(* CODESYS project SkyP_crashtest

Project tree, tasks and I/O mapping:
  Device : CODESYS Control for Linux SL, CODESYS, order no. 2302000005, version 4.13.0.0
    Ethernet : Ethernet, CODESYS, version 4.2.0.0
        settings: IPAddress = [192,168,1,12]; SubnetMask = [255,255,255,0]; GatewayAddress = [192,168,1,1]; MACAddress = [16#00,16#E0,16#4F,16#68,16#EC,16#5C]; NetworkInterfaceName = 'eno1'; NetworkInterfaceName = "eno1"; SaveCommunicationSettings = FALSE; IPAddress = [192,168,0,2]; SubnetMask = [255,255,255,0]; GatewayAddress = [0,0,0,0]
      Modbus_TCP_Master : Modbus TCP Client, CODESYS, version 4.4.0.0
          settings: AutoReconnect = TRUE
        Modbus_TCP_Slave_AC1 : Modbus TCP Slave, 3S - Smart Software Solutions GmbH, version 4.1.0.0
            settings: Unit-ID = 255; IPAddress = [192, 168, 0, 51]; Channel 0.Function Code = 3; Channel 0.Read Offset = 16#0000; Channel 0.Read Length = 124; Channel 0.Write Offset = 0; Channel 0.Write Length = 0; Channel 0.Cycle Time = 100; Channel 1.Function Code = 3; Channel 1.Read Offset = 16#007C; Channel 1.Read Length = 124; Channel 1.Write Offset = 0; Channel 1.Write Length = 0; Channel 1.Cycle Time = 100; Channel 2.Function Code = 3; Channel 2.Read Offset = 16#00F8; Channel 2.Read Length = 124; Channel 2.Write Offset = 0; Channel 2.Write Length = 0; Channel 2.Cycle Time = 100; Channel 3.Function Code = 16; Channel 3.Read Offset = 0; Channel 3.Read Length = 0; Channel 3.Write Offset = 16#0114; Channel 3.Write Length = 4; Channel 3.Cycle Time = 100
            input  Application.Chiller_1.modbus_var_1000 : ARRAY[0..123] OF WORD  // Channel 0
            input  Application.Chiller_1.modbus_var_1001 : ARRAY[0..123] OF WORD  // Channel 1
            input  Application.Chiller_1.modbus_var_1002 : ARRAY[0..123] OF WORD  // Channel 2
            output Application.Chiller_1.modbus_var_1002[276] : WORD  // Channel 3.Channel 3
            output Application.Chiller_1.modbus_var_1002[277] : WORD  // Channel 3.Channel 3
            output Application.Chiller_1.modbus_var_1002[278] : WORD  // Channel 3.Channel 3
            output Application.Chiller_1.modbus_var_1002[279] : WORD  // Channel 3.Channel 3
            unmapped channels: Channel 3
        Modbus_TCP_Slave_AC2 : Modbus TCP Slave, 3S - Smart Software Solutions GmbH, version 4.1.0.0
            settings: Unit-ID = 255; IPAddress = [192, 168, 0, 52]; Channel 0.Function Code = 3; Channel 0.Read Offset = 16#0000; Channel 0.Read Length = 124; Channel 0.Write Offset = 0; Channel 0.Write Length = 0; Channel 0.Cycle Time = 100; Channel 1.Function Code = 3; Channel 1.Read Offset = 16#007C; Channel 1.Read Length = 124; Channel 1.Write Offset = 0; Channel 1.Write Length = 0; Channel 1.Cycle Time = 100; Channel 2.Function Code = 3; Channel 2.Read Offset = 16#00F8; Channel 2.Read Length = 124; Channel 2.Write Offset = 0; Channel 2.Write Length = 0; Channel 2.Cycle Time = 100; Channel 3.Function Code = 16; Channel 3.Read Offset = 0; Channel 3.Read Length = 0; Channel 3.Write Offset = 16#0114; Channel 3.Write Length = 4; Channel 3.Cycle Time = 100
            input  Application.Chiller_2.modbus_var_1000 : ARRAY[0..123] OF WORD  // Channel 0
            input  Application.Chiller_2.modbus_var_1001 : ARRAY[0..123] OF WORD  // Channel 1
            input  Application.Chiller_2.modbus_var_1002 : ARRAY[0..123] OF WORD  // Channel 2
            output Application.Chiller_2.modbus_var_1002[276] : WORD  // Channel 3.Channel 3
            output Application.Chiller_2.modbus_var_1002[277] : WORD  // Channel 3.Channel 3
            output Application.Chiller_2.modbus_var_1002[278] : WORD  // Channel 3.Channel 3
            output Application.Chiller_2.modbus_var_1002[279] : WORD  // Channel 3.Channel 3
            unmapped channels: Channel 3
        Modbus_TCP_Slave_AC3 : Modbus TCP Slave, 3S - Smart Software Solutions GmbH, version 4.1.0.0
            settings: Unit-ID = 255; IPAddress = [192, 168, 0, 53]; Channel 0.Function Code = 3; Channel 0.Read Offset = 16#0000; Channel 0.Read Length = 124; Channel 0.Write Offset = 0; Channel 0.Write Length = 0; Channel 0.Cycle Time = 100; Channel 1.Function Code = 3; Channel 1.Read Offset = 16#007C; Channel 1.Read Length = 124; Channel 1.Write Offset = 0; Channel 1.Write Length = 0; Channel 1.Cycle Time = 100; Channel 2.Function Code = 3; Channel 2.Read Offset = 16#00F8; Channel 2.Read Length = 124; Channel 2.Write Offset = 0; Channel 2.Write Length = 0; Channel 2.Cycle Time = 100; Channel 3.Function Code = 16; Channel 3.Read Offset = 0; Channel 3.Read Length = 0; Channel 3.Write Offset = 16#0114; Channel 3.Write Length = 4; Channel 3.Cycle Time = 100
            input  Application.Chiller_3.modbus_var_1000 : ARRAY[0..123] OF WORD  // Channel 0
            input  Application.Chiller_3.modbus_var_1001 : ARRAY[0..123] OF WORD  // Channel 1
            input  Application.Chiller_3.modbus_var_1002 : ARRAY[0..123] OF WORD  // Channel 2
            output Application.Chiller_3.modbus_var_1002[276] : WORD  // Channel 3.Channel 3
            output Application.Chiller_3.modbus_var_1002[277] : WORD  // Channel 3.Channel 3
            output Application.Chiller_3.modbus_var_1002[278] : WORD  // Channel 3.Channel 3
            output Application.Chiller_3.modbus_var_1002[279] : WORD  // Channel 3.Channel 3
            unmapped channels: Channel 3
        Modbus_TCP_Slave_AC4 : Modbus TCP Slave, 3S - Smart Software Solutions GmbH, version 4.1.0.0
            settings: Unit-ID = 255; IPAddress = [192, 168, 0, 54]; Channel 0.Function Code = 3; Channel 0.Read Offset = 16#0000; Channel 0.Read Length = 124; Channel 0.Write Offset = 0; Channel 0.Write Length = 0; Channel 0.Cycle Time = 100; Channel 1.Function Code = 3; Channel 1.Read Offset = 16#007C; Channel 1.Read Length = 124; Channel 1.Write Offset = 0; Channel 1.Write Length = 0; Channel 1.Cycle Time = 100; Channel 2.Function Code = 3; Channel 2.Read Offset = 16#00F8; Channel 2.Read Length = 124; Channel 2.Write Offset = 0; Channel 2.Write Length = 0; Channel 2.Cycle Time = 100; Channel 3.Function Code = 16; Channel 3.Read Offset = 0; Channel 3.Read Length = 0; Channel 3.Write Offset = 16#0114; Channel 3.Write Length = 4; Channel 3.Cycle Time = 100
            input  Application.Chiller_4.modbus_var_1000 : ARRAY[0..123] OF WORD  // Channel 0
            input  Application.Chiller_4.modbus_var_1001 : ARRAY[0..123] OF WORD  // Channel 1
            input  Application.Chiller_4.modbus_var_1002 : ARRAY[0..123] OF WORD  // Channel 2
            output Application.Chiller_4.modbus_var_1002[276] : WORD  // Channel 3.Channel 3
            output Application.Chiller_4.modbus_var_1002[277] : WORD  // Channel 3.Channel 3
            output Application.Chiller_4.modbus_var_1002[278] : WORD  // Channel 3.Channel 3
            output Application.Chiller_4.modbus_var_1002[279] : WORD  // Channel 3.Channel 3
            unmapped channels: Channel 3
        Modbus_TCP_Slave_AC5 : Modbus TCP Slave, 3S - Smart Software Solutions GmbH, version 4.1.0.0
            settings: Unit-ID = 255; IPAddress = [192, 168, 0, 55]; Channel 0.Function Code = 3; Channel 0.Read Offset = 16#0000; Channel 0.Read Length = 124; Channel 0.Write Offset = 0; Channel 0.Write Length = 0; Channel 0.Cycle Time = 100; Channel 1.Function Code = 3; Channel 1.Read Offset = 16#007C; Channel 1.Read Length = 124; Channel 1.Write Offset = 0; Channel 1.Write Length = 0; Channel 1.Cycle Time = 100; Channel 2.Function Code = 3; Channel 2.Read Offset = 16#00F8; Channel 2.Read Length = 124; Channel 2.Write Offset = 0; Channel 2.Write Length = 0; Channel 2.Cycle Time = 100; Channel 3.Function Code = 16; Channel 3.Read Offset = 0; Channel 3.Read Length = 0; Channel 3.Write Offset = 16#0114; Channel 3.Write Length = 4; Channel 3.Cycle Time = 100
            input  Application.Chiller_5.modbus_var_1000 : ARRAY[0..123] OF WORD  // Channel 0
            input  Application.Chiller_5.modbus_var_1001 : ARRAY[0..123] OF WORD  // Channel 1
            input  Application.Chiller_5.modbus_var_1002 : ARRAY[0..123] OF WORD  // Channel 2
            output Application.Chiller_5.modbus_var_1002[276] : WORD  // Channel 3.Channel 3
            output Application.Chiller_5.modbus_var_1002[277] : WORD  // Channel 3.Channel 3
            output Application.Chiller_5.modbus_var_1002[278] : WORD  // Channel 3.Channel 3
            output Application.Chiller_5.modbus_var_1002[279] : WORD  // Channel 3.Channel 3
            unmapped channels: Channel 3
  libraries: CmpBitmapPool, 3.5.17.0 (System); AC_DataLog, 3.5.16.0 (3S - Smart Software Solutions GmbH)
  5ce3da45-db07-42e7-a21c-a00fff4ed8f6|C:\Users\Technician\Desktop\Images\Chiller\Compressor2.png
  5ce3da45-db07-42e7-a21c-a00fff4ed8f6|C:\Users\Technician\Desktop\Images\Chiller\Ejector.png
  5ce3da45-db07-42e7-a21c-a00fff4ed8f6|C:\Users\Technician\Desktop\Images\Chiller\Evaporator2.png
  5ce3da45-db07-42e7-a21c-a00fff4ed8f6|C:\Users\Technician\Desktop\Images\Chiller\OilFilter.png
  5ce3da45-db07-42e7-a21c-a00fff4ed8f6|C:\Users\Technician\Desktop\Images\Chiller\OilReceiver.png
  5ce3da45-db07-42e7-a21c-a00fff4ed8f6|C:\Users\Technician\Desktop\Images\Div bilder\Arrow black down.png
  5ce3da45-db07-42e7-a21c-a00fff4ed8f6|C:\Users\Technician\Desktop\Images\Div bilder\Arrow black left.png
  5ce3da45-db07-42e7-a21c-a00fff4ed8f6|C:\Users\Technician\Desktop\Images\Div bilder\Arrow black right.png
  5ce3da45-db07-42e7-a21c-a00fff4ed8f6|C:\Users\Technician\Desktop\Images\Div bilder\Arrow black up.png
  5ce3da45-db07-42e7-a21c-a00fff4ed8f6|C:\Users\Technician\Desktop\Images\Div bilder\Arrow gray right.png
  5ce3da45-db07-42e7-a21c-a00fff4ed8f6|C:\Users\Technician\Desktop\Images\Div bilder\Arrow red up.png
  5ce3da45-db07-42e7-a21c-a00fff4ed8f6|C:\Users\Technician\Desktop\Images\HeatExchanger\OilHeatExchanger.png
  5ce3da45-db07-42e7-a21c-a00fff4ed8f6|C:\Users\Technician\Desktop\Images\Menu\CalendarIcon.png
  5ce3da45-db07-42e7-a21c-a00fff4ed8f6|C:\Users\Technician\Desktop\Images\Menu\Logo-Carnival.png
  5ce3da45-db07-42e7-a21c-a00fff4ed8f6|C:\Users\Technician\Desktop\Images\Menu\MenuTrends.png
  5ce3da45-db07-42e7-a21c-a00fff4ed8f6|C:\Users\Technician\Desktop\Images\New\VSD_rev2.png
  5ce3da45-db07-42e7-a21c-a00fff4ed8f6|C:\Users\Technician\Desktop\Images\Pipes\PipeBlack_1_Horizontal.png
  5ce3da45-db07-42e7-a21c-a00fff4ed8f6|C:\Users\Technician\Desktop\Images\Pipes\PipeBlack_1_LD.png
  5ce3da45-db07-42e7-a21c-a00fff4ed8f6|C:\Users\Technician\Desktop\Images\Pipes\PipeBlack_1_LU.png
  5ce3da45-db07-42e7-a21c-a00fff4ed8f6|C:\Users\Technician\Desktop\Images\Pipes\PipeBlack_1_RD.png
  5ce3da45-db07-42e7-a21c-a00fff4ed8f6|C:\Users\Technician\Desktop\Images\Pipes\PipeBlack_1_RU.png
  5ce3da45-db07-42e7-a21c-a00fff4ed8f6|C:\Users\Technician\Desktop\Images\Pipes\PipeBlack_1_Vertical.png
  5ce3da45-db07-42e7-a21c-a00fff4ed8f6|C:\Users\Technician\Desktop\Images\Pipes\PipeBlack_1S_H_Faded.png
  5ce3da45-db07-42e7-a21c-a00fff4ed8f6|C:\Users\Technician\Desktop\Images\Ships\Norwegian Prima.jpg
  5ce3da45-db07-42e7-a21c-a00fff4ed8f6|C:\Users\Technician\Desktop\Images\Ships\SkyPrincess.jpg
  5ce3da45-db07-42e7-a21c-a00fff4ed8f6|C:\Users\Technician\Desktop\Images\Valves\RegValve.png
  AC_GENERATOR_DATA
  DataLogManager
    Channels for DataLog (DataLogChannels)
      DataLogChannel_1
        A storage module. (DataLogStorage)
        DataLogStorage_CSV
      DataLogChannel_2
        A storage module. (DataLogStorage)
        DataLogStorage_CSV
      DataLogChannel_3
        A storage module. (DataLogStorage)
        DataLogStorage_CSV
      DataLogChannel_4
        A storage module. (DataLogStorage)
        DataLogStorage_CSV
      DataLogChannel_5
        A storage module. (DataLogStorage)
        DataLogStorage_CSV
      DataLogChannel
        A storage module. (DataLogStorage)
        DataLogStorage_CSV
  text list GlobalTextList
  PersistenceManager
    Channels (pChannels)
      PersistenceChannel
  Alarm Configuration
  visualisation Alarm_list
  program BlinkingAlarm [CFC]
  program Calculus [ST]
  visualisation Chiller1Menu
  visualisation Chiller2Menu
  visualisation Chiller3Menu
  visualisation Chiller4Menu
  visualisation Chiller5Menu
  program Chiller_1 [ST]
  visualisation Chiller_1_Alarm
  visualisation Chiller_1_Flow_Diagram
  visualisation Chiller_1_Oil
  visualisation Chiller_1_Trip
  visualisation Chiller_1_Values
  visualisation Chiller_2_Alarm
  program Chiller_2 [ST]
  visualisation Chiller_2_Flow_Diagram
  visualisation Chiller_2_Oil
  visualisation Chiller_2_Trip
  visualisation Chiller_2_Values
  visualisation Chiller_2_VFD
  program Chiller_3 [ST]
  visualisation Chiller_3_Alarm
  visualisation Chiller_3_Flow_Diagram
  visualisation Chiller_3_Oil
  program Chiller_4 [ST]
  program Chiller_5 [ST]
  text list Chiller_trendvalues
  text list Chiller_VSD_trendvalues
  program csvRead [CFC]
  global variables GVL
  visualisation Homepage
  text list TextList_Local_IAMCS
*)

// GVL
{attribute 'qualified_only'}
VAR_GLOBAL
	COPcalc_data	: ARRAY[0..2, 0..320] OF STRING(100);
	calc_data		: ARRAY[0..8, 0..80] OF STRING(100) ;
	{attribute 'ac_persist' := 'PersistenceChannel'}
	saCOPDataArray			: ARRAY[0..2, 0..320] OF STRING(100);
	{attribute 'ac_persist' := 'PersistenceChannel'}
	saDataArray			: ARRAY[0..8, 0..80] OF STRING(100);
	{attribute 'ac_persist' := 'PersistenceChannel'}
	saDataArray1			: ARRAY[0..8, 0..80] OF STRING(100);
	{attribute 'ac_persist' := 'PersistenceChannel'}
	saDataArray2		: ARRAY[0..8, 0..80] OF STRING(100);
	{attribute 'ac_persist' := 'PersistenceChannel'}
	saDataArray3		: ARRAY[0..8, 0..80] OF STRING(100);
	initRead : BOOL;
	xRead : BOOL;
	xRead1 : BOOL;
	xRead2 : BOOL;
	xRead3 : BOOL;
	xReadCOP : BOOL := FALSE;
	startUp : BOOL;
	presstimer  : TON;
	presstimer2 : TON;
	presstimer3 : TON;
	presstimer4 : TON;
	presstimer5 : TON;
	delaytimer  : TON;
	starttimer1 : BOOL := FALSE  ;
	starttimer2 : BOOL := FALSE  ;
	starttimer3 : BOOL := FALSE  ;
	starttimer4 : BOOL := FALSE  ;
	starttimer5 : BOOL := FALSE  ;
	startdelaytimer : BOOL := FALSE ;
	Startonce : BOOL := FALSE ;
	Startsecond : BOOL := FALSE ;
	{attribute 'ac_persist' := 'PersistenceChannel'}
	PIexpireDate : DATE_AND_TIME := DT#2026-01-31-00:00:00;
	CurrentDate : DATE_AND_TIME ;

END_VAR

// BlinkingAlarm
PROGRAM BlinkingAlarm
VAR
	TimeOn: TIME:= T#1S;
	TimeOff: TIME:= T#1S;
	Alarm: BOOL;
	TurnOn: BOOL;
		
	Blink_0: BLINK;
	
END_VAR
VAR // added by the converter: edge detectors and wires of the graphical bodies
    _w1, _w2 : BOOL;
END_VAR

TurnOn := _w1;
_w1 := not.Sequence.Alarm_sequence OR not.Chiller_1.Unit_alarm OR not.Chiller_1.Unit_trip OR not.Chiller_2.Unit_alarm OR not.Chiller_2.Unit_trip OR not.Chiller_3.Unit_alarm OR not.Chiller_3.Unit_trip OR not.Chiller_4.Unit_alarm OR not.Chiller_4.Unit_trip OR not.Chiller_5.Unit_alarm OR not.Chiller_5.Unit_trip;
_w2 := TurnOn AND Blink_0.OUT;
Blink_0(ENABLE := TurnOn, TIMELOW := TimeOff, TIMEHIGH := TimeOn); // BLINK
Alarm := _w2;

END_PROGRAM

// Chiller_5
PROGRAM Chiller_5
VAR

timer2 : standard.ton ;
{attribute 'ac_datalog_set_default_group' := 'DataLogChannel_5'}
instStruct : LogStruct;


modbus_var : ARRAY[0..100] OF INT;
modbus_var_1000 : ARRAY[0..123] OF WORD;
modbus_var_1001 : ARRAY[124..247] OF WORD;
modbus_var_1002 : ARRAY[248..371] OF WORD;
{attribute 'ac_datalog_hysteresis' := '0.2'}
{attribute 'ac_datalog' := 'DataLogChannel_5'}
Temp_chilled_medium_out : REAL;
{attribute 'ac_datalog_hysteresis' := '0.2'}
{attribute 'ac_datalog' := 'DataLogChannel_5'}
Temp_chilled_medium_in : REAL;
{attribute 'ac_datalog_hysteresis' := '0.2'}
{attribute 'ac_datalog' := 'DataLogChannel_5'}
Temp_water_inlet_cond : REAL;
{attribute 'ac_datalog_hysteresis' := '0.2'}
{attribute 'ac_datalog' := 'DataLogChannel_5'}
Press_suction_compr : REAL;
{attribute 'ac_datalog_hysteresis' := '0.5'}
{attribute 'ac_datalog' := 'DataLogChannel_5'}
Press_discharge_compr : REAL;
{attribute 'ac_datalog_hysteresis' := '0.5'}
{attribute 'ac_datalog' := 'DataLogChannel_5'}
Press_oil_receiver : REAL;
{attribute 'ac_datalog_hysteresis' := '0.5'}
{attribute 'ac_datalog' := 'DataLogChannel_5'}
Press_oil_compr : REAL;
{attribute 'ac_datalog_hysteresis' := '0.4'}
{attribute 'ac_datalog' := 'DataLogChannel_5'}
Temp_discharge : REAL;
{attribute 'ac_datalog_hysteresis' := '0.5'}
{attribute 'ac_datalog' := 'DataLogChannel_5'}
Oil_temp_receiver : REAL;
{attribute 'ac_datalog_hysteresis' := '0.5'}
{attribute 'ac_datalog' := 'DataLogChannel_5'}
Max_motor_temp : REAL;
{attribute 'ac_datalog_hysteresis' := '0.2'}
{attribute 'ac_datalog' := 'DataLogChannel_5'}
Temp_motor_bearing_DE : REAL;
{attribute 'ac_datalog_hysteresis' := '0.2'}
{attribute 'ac_datalog' := 'DataLogChannel_5'}
Temp_motor_bearing_NDE : REAL;
{attribute 'ac_datalog_hysteresis' := '4'}
{attribute 'ac_datalog' := 'DataLogChannel_5'}
Motor_current : REAL;
{attribute 'ac_datalog_hysteresis' := '50'}
{attribute 'ac_datalog' := 'DataLogChannel_5'}
Running_hours_comp_unscaled : WORD;
{attribute 'ac_datalog_hysteresis' := '50'}
{attribute 'ac_datalog' := 'DataLogChannel_5'}
Running_hours_oil_pump_unscaled : WORD;
{attribute 'ac_datalog' := 'DataLogChannel_5'}
Anti_recycle_time : REAL;
{attribute 'ac_datalog_hysteresis' := '2'}
{attribute 'ac_datalog' := 'DataLogChannel_5'}
Feedback_compressor : REAL;
{attribute 'ac_datalog_hysteresis' := '0.2'}
{attribute 'ac_datalog' := 'DataLogChannel_5'}
Oil_diff_pressure : REAL;
{attribute 'ac_datalog_hysteresis' := '0.3'}
{attribute 'ac_datalog' := 'DataLogChannel_5'}
Suction_saturated_temp : REAL;
{attribute 'ac_datalog_hysteresis' := '0.2'}
{attribute 'ac_datalog' := 'DataLogChannel_5'}
Discharge_saturated_temp : REAL;
{attribute 'ac_datalog_hysteresis' := '0.2'}
{attribute 'ac_datalog' := 'DataLogChannel_5'}
Temp_water_outlet_cond : REAL;
{attribute 'ac_datalog_hysteresis' := '0.2'}
{attribute 'ac_datalog' := 'DataLogChannel_5'}
Temp_motor_wind_R : REAL;
{attribute 'ac_datalog_hysteresis' := '0.2'}
{attribute 'ac_datalog' := 'DataLogChannel_5'}
Temp_motor_wind_S : REAL;
{attribute 'ac_datalog_hysteresis' := '0.2'}
{attribute 'ac_datalog' := 'DataLogChannel_5'}
Temp_motor_wind_T : REAL;
{attribute 'ac_datalog_hysteresis' := '0.2'}
{attribute 'ac_datalog' := 'DataLogChannel_5'}
Temp_motor_air : REAL;
{attribute 'ac_datalog_hysteresis' := '0.04'}
{attribute 'ac_datalog' := 'DataLogChannel_5'}
dP_CW : REAL;
{attribute 'ac_datalog_hysteresis' := '0.04'}
{attribute 'ac_datalog' := 'DataLogChannel_5'}
dP_SW : REAL;
{attribute 'ac_datalog_hysteresis' := '4'}
{attribute 'ac_datalog' := 'DataLogChannel_5'}
Chiller_capacity : REAL;
{attribute 'ac_datalog_hysteresis' := '2'}
{attribute 'ac_datalog' := 'DataLogChannel_5'}
Temp_oil_inlet_compr : REAL;
Spare : REAL;
{attribute 'ac_datalog_hysteresis' := '2'}
{attribute 'ac_datalog' := 'DataLogChannel_5'}
SP_CW_controller : REAL;
{attribute 'ac_datalog_hysteresis' := '2'}
{attribute 'ac_datalog' := 'DataLogChannel_5'}
Setpoint_oil_pump : REAL;
{attribute 'ac_datalog_hysteresis' := '0.02'}
{attribute 'ac_datalog' := 'DataLogChannel_5'}
Thrust_bearing_position : REAL;
{attribute 'ac_datalog_hysteresis' := '50'}
{attribute 'ac_datalog' := 'DataLogChannel_5'}
Oil_pump_running_hours : REAL;
{attribute 'ac_datalog_hysteresis' := '5'}
{attribute 'ac_datalog' := 'DataLogChannel_5'}
Liquid_level_condenser : REAL;
{attribute 'ac_datalog_hysteresis' := '0.05'}
{attribute 'ac_datalog' := 'DataLogChannel_5'}
Oil_Filter_Drop : REAL; 
{attribute 'ac_datalog_hysteresis' := '2'}
{attribute 'ac_datalog' := 'DataLogChannel_5'}
Proximitor_thrust_pos : REAL;
{attribute 'ac_datalog_hysteresis' := '0.4'}
{attribute 'ac_datalog' := 'DataLogChannel_5'}
Press_chilled_medium_in : REAL;
{attribute 'ac_datalog_hysteresis' := '0.2'}
{attribute 'ac_datalog' := 'DataLogChannel_5'}
Press_water_cond_out : REAL;
{attribute 'ac_datalog_hysteresis' := '0.02'}
{attribute 'ac_datalog' := 'DataLogChannel_5'}
Feedback_sea_water_valve : REAL;
{attribute 'ac_datalog_hysteresis' := '1'}
{attribute 'ac_datalog' := 'DataLogChannel_5'}
Oil_pressure_before_filter : REAL;
{attribute 'ac_datalog_hysteresis' := '0.2'}
{attribute 'ac_datalog' := 'DataLogChannel_5'}
Trafo_winding_temp : REAL;
{attribute 'ac_datalog_hysteresis' := '1'}
{attribute 'ac_datalog' := 'DataLogChannel_5'}
Feedback_VGD : REAL;
{attribute 'ac_datalog_hysteresis' := '4'}
{attribute 'ac_datalog' := 'DataLogChannel_5'}
Feedback_liquid_valve : REAL;
{attribute 'ac_datalog_hysteresis' := '3'}
{attribute 'ac_datalog' := 'DataLogChannel_5'}
Feedback_HGV : REAL;
{attribute 'ac_datalog_hysteresis' := '2'}
{attribute 'ac_datalog' := 'DataLogChannel_5'}
Discharge_superheat : REAL;
{attribute 'ac_datalog_hysteresis' := '0.6'}
{attribute 'ac_datalog' := 'DataLogChannel_5'}
Frequency_oil_pump : REAL;
{attribute 'ac_datalog_hysteresis' := '3'}
{attribute 'ac_datalog' := 'DataLogChannel_5'}
Hot_gas_valve_output : REAL;
{attribute 'ac_datalog_hysteresis' := '2'}
{attribute 'ac_datalog' := 'DataLogChannel_5'}
Control_signal_unit_d : REAL;
{attribute 'ac_datalog_hysteresis' := '2'}
{attribute 'ac_datalog' := 'DataLogChannel_5'}
Stall_detector : REAL;
{attribute 'ac_datalog_hysteresis' := '0.2'}
{attribute 'ac_datalog' := 'DataLogChannel_5'}
SP_MC_controller : REAL;
{attribute 'ac_datalog_hysteresis' := '2'}
{attribute 'ac_datalog' := 'DataLogChannel_5'}
Prerotary_output : REAL;
{attribute 'ac_datalog_hysteresis' := '2'}
{attribute 'ac_datalog' := 'DataLogChannel_5'}
VGD_output : REAL;
{attribute 'ac_datalog_hysteresis' := '2'}
{attribute 'ac_datalog' := 'DataLogChannel_5'}
SP_PID_compressor : REAL;
{attribute 'ac_datalog_hysteresis' := '2'}
{attribute 'ac_datalog' := 'DataLogChannel_5'}
Output_PID_suction : REAL;
{attribute 'ac_datalog_hysteresis' := '2'}
{attribute 'ac_datalog' := 'DataLogChannel_5'}
Output_PID_discharge : REAL;
{attribute 'ac_datalog_hysteresis' := '2'}
{attribute 'ac_datalog' := 'DataLogChannel_5'}
Output_PID_motor : REAL;
{attribute 'ac_datalog_hysteresis' := '2'}
{attribute 'ac_datalog' := 'DataLogChannel_5'}
Output_PID_superheat : REAL;
{attribute 'ac_datalog_hysteresis' := '2'}
{attribute 'ac_datalog' := 'DataLogChannel_5'}
SP_control : REAL;
{attribute 'ac_datalog_hysteresis' := '2'}
{attribute 'ac_datalog' := 'DataLogChannel_5'}
Unit_control_signal : REAL;
{attribute 'ac_datalog_hysteresis' := '2'}
{attribute 'ac_datalog' := 'DataLogChannel_5'}
Feedback_PRV : REAL;
{attribute 'ac_datalog_hysteresis' := '0.3'}
{attribute 'ac_datalog' := 'DataLogChannel_5'}
Theta_out : REAL;
{attribute 'ac_datalog_hysteresis' := '50'}
{attribute 'ac_datalog' := 'DataLogChannel_5'}
Alarm_limit_stall_count_unscaled : WORD;
{attribute 'ac_datalog_hysteresis' := '50'}
{attribute 'ac_datalog' := 'DataLogChannel_5'}
Alarm_limit_stall_count : REAL;
{attribute 'ac_datalog_hysteresis' := '2'}
{attribute 'ac_datalog' := 'DataLogChannel_5'}
Stall_ramp : REAL;
Min_allowed_PRVposition : REAL;
Number_of_starts : REAL;
SP_oil_pressure : REAL;
{attribute 'ac_datalog_hysteresis' := '2'}
{attribute 'ac_datalog' := 'DataLogChannel_5'}
Setpoint_conv_oil_pump : REAL;
Days_above_stall_limit : REAL;
Hrs_above_stall_limit : REAL;
Min_above_stall_limit : REAL;
Sec_above_stall_limit : REAL;
{attribute 'ac_datalog_hysteresis' := '2'}
{attribute 'ac_datalog' := 'DataLogChannel_5'}
SP_cond_press : REAL;
{attribute 'ac_datalog_hysteresis' := '2'}
{attribute 'ac_datalog' := 'DataLogChannel_5'}
SP_PID_Level : REAL;
{attribute 'ac_datalog_hysteresis' := '2'}
{attribute 'ac_datalog' := 'DataLogChannel_5'}
Control_signal_SW_valve : REAL;
{attribute 'ac_datalog_hysteresis' := '4'}
{attribute 'ac_datalog' := 'DataLogChannel_5'}
Liquid_valve_output : REAL;
{attribute 'ac_datalog_hysteresis' := '0.2'}
{attribute 'ac_datalog' := 'DataLogChannel_5'}
SP_PID_seawater : REAL;
{attribute 'ac_datalog_hysteresis' := '4'}
{attribute 'ac_datalog' := 'DataLogChannel_5'}
Chiller_capacity_t1 : REAL;
{attribute 'ac_datalog_hysteresis' := '2'}
{attribute 'ac_datalog' := 'DataLogChannel_5'}
SW_pump_speed_order : REAL;
{attribute 'ac_datalog_hysteresis' := '0.4'}
{attribute 'ac_datalog' := 'DataLogChannel_5'}
Press_chilled_medium_out : REAL;
{attribute 'ac_datalog_hysteresis' := '50'}
{attribute 'ac_datalog' := 'DataLogChannel_5'}
Running_hours_compressormotor : REAL;
{attribute 'ac_datalog_hysteresis' := '0.2'}
{attribute 'ac_datalog' := 'DataLogChannel_5'}
Press_water_cond_inlet : REAL;
Speed_feedback_VFD : REAL;
Order_VFD_perc : REAL;
Order_VFD_Hz : REAL;
{attribute 'ac_datalog_hysteresis' := '2'}
{attribute 'ac_datalog' := 'DataLogChannel_5'}
Temp_trafo_wind_U : REAL;
{attribute 'ac_datalog_hysteresis' := '0.2'}
{attribute 'ac_datalog' := 'DataLogChannel_5'}
Temp_trafo_wind_V : REAL;
{attribute 'ac_datalog_hysteresis' := '0.2'}
{attribute 'ac_datalog' := 'DataLogChannel_5'}
Temp_trafo_wind_W : REAL;
Opt_speed_VFD_perc : REAL;
Opt_speed_VFD_Hz : REAL;
Surge_counter_VFD : REAL;
Spare_4 : REAL;
Spare_3 : REAL;
Spare_2 : REAL;
Spare_0 : REAL;
Vibration_compressor_DE: REAL;
Vibration_compressor_NDE: REAL;
Feedback_seawater_valve_overboard : REAL;
Feedback_seawater_valve_bypass : REAL;
CW_flow_m3: REAL;
SW_flow_m3: REAL;
Max_motor_wind_temp: REAL;
Order_SWW_overboard: REAL;
Order_SWW_bypass: REAL;
{attribute 'ac_datalog_hysteresis' := '0.4'}
{attribute 'ac_datalog' := 'DataLogChannel'}
COP_chiller_mech : REAL ;
{attribute 'ac_datalog_hysteresis' := '10'}
{attribute 'ac_datalog' := 'DataLogChannel'}
P2_mot_1_kW : REAL ;
{attribute 'ac_datalog_hysteresis' := '20'}
{attribute 'ac_datalog' := 'DataLogChannel'}
P1_motor_kW : REAL ;
{attribute 'ac_datalog_hysteresis' := '0.4'}
{attribute 'ac_datalog' := 'DataLogChannel'}
COP_chiller_ele : REAL ;
{attribute 'ac_datalog_hysteresis' := '0.2'}
{attribute 'ac_datalog' := 'DataLogChannel'}
PI_chiller : REAL ;
{attribute 'ac_datalog_hysteresis' := '40'}
{attribute 'ac_datalog' := 'DataLogChannel'}
Wasted_energy_kW : REAL ;
{attribute 'ac_datalog_hysteresis' := '200'}
{attribute 'ac_datalog' := 'DataLogChannel'}
Chiller_capacity_kW : REAL;
Thrust_bearing_ref_min : REAL ;
Thrust_bearing_ref_max : REAL ;
Thrust_bearing_ref : REAL ;
Q2_chillerMWh : REAL ;
Chiller_P1_MWh : REAL ;
Cal_date_MMYY : REAL ;
Chiller_P2_MWh : REAL ;
Liquid_line_temp : REAL ;
VFD_motor_current : REAL ;
Feedback_liquid_valve_raw : REAL ;
Feedback_VGD_raw : REAL ;
Feedback_PRV_raw : REAL ;
Feedback_HGV_raw : REAL ;
Feedback_seawater_valve_overboard_raw : REAL ;
Feedback_seawater_valve_bypass_raw : REAL ;
SP_cond_press_limit : REAL ;
SP_evap_press_limit : REAL ;
SP_discharge_superheat_limit : REAL ;
VFD_min_allowed_frequence : REAL ;
VFD_min_allowed_speed : REAL ;
CW_Pump_Speed_SP : REAL;

Trip_BITs_0_to_15 : WORD;
Trip_BITs_16_to_31: WORD;
Trip_BITs_32_to_47: WORD;
Trip_BITs_48_to_63: WORD;
Trip_BITs_64_to_79: WORD;
Trip_BITs_80_to_95: WORD;
Trip_BITs_96_to_121: WORD;
Trip_BITs_122_to_137: WORD;
Trip_BITs_138_to_153: WORD;
Trip_BITs_154_to_169: WORD;
Trip_BITs_170_to_185: WORD;
Trip_BITs_186_to_201: WORD;


Alarm_BITs_0_to_15: WORD;
Alarm_BITs_16_to_31: WORD;
Alarm_BITs_32_to_47: WORD;
Alarm_BITs_48_to_63: WORD;
Alarm_BITs_64_to_79: WORD;
Status_BITs_0_to_15 : WORD;
Status_BITs_16_to_31 : WORD;
Status_BITs_32_to_47: WORD;
Status_BITs_48_to_63: WORD;
Status_BITs_64_to_79: WORD;
Status_BITs_80_to_95: WORD;




DIStatusbits_0_to_15 : WORD;
DIStatusbits_16_to_31: WORD;

DOStatusbits_16_to_31: WORD;
DOStatusbits_32_to_47: WORD;

T_Overload_compressor_motor : BOOL;
T_Compressor_running_failure : BOOL;

T_Low_oil_flow : BOOL;
T_Overload_oil_pump_motor : BOOL;
T_Oil_pump_running_failure : BOOL;
T_Low_oil_flow_trip : BOOL;
T_High_temp_oil_receiver : BOOL;
T_Low_temp_oil_receiver : BOOL;
T_Low_suction_pressure : BOOL;
T_High_suction_pressure : BOOL;
T_High_discharge_pressure : BOOL;
T_Low_discharge_pressure : BOOL;
T_High_discharge_temp : BOOL;
T_Low_oil_diff_pressure : BOOL;
T_High_diff_oil_pressure : BOOL;
T_Starting_to_long : BOOL;
T_Surge_detection : BOOL;
T_Comp_thrust_bearing_position : BOOL;
Spare_trip_1 : BOOL;
T_Chilled_pump_run_failure : BOOL;
T_Sea_water_pump_run_failure : BOOL;
T_Low_chilled_medium_flow : BOOL;
T_High_chilled_medium_flow : BOOL;
T_Low_condenser_flow : BOOL;
T_High_condenser_flow : BOOL;
T_Emergency_stop : BOOL;
T_High_comp_mot_DE_bear_temp : BOOL;
T_High_comp_mot_NDE_bear_temp : BOOL;
T_High_motor_air_temp : BOOL;
T_Comp_motor_leak_detection : BOOL;
T_High_comp_mot_DE_bear_vib : BOOL;
T_High_comp_mot_NDE_bear_Vib : BOOL;
Spare_trip_2 : BOOL;
T_Rotating_stall_trip : BOOL;
T_Analog_inputs : BOOL;
T_Feedback_CW_valve : BOOL;
T_Low_oil_diff_press_prelub : BOOL;
T_Low_oil_diff_press_standstil : BOOL;

T_Spare_3 : BOOL;
T_Spare_4 : BOOL;
T_Spare_5 : BOOL;
T_Spare_6 : BOOL;
T_Spare_7 : BOOL;
T_Spare_8 : BOOL;
T_High_temp_oil_inlet_comp : BOOL;
T_Comp_motor_power_loss : BOOL;
Spare_trip_3 : BOOL;
T_Cathodic_protect_sys_alarm : BOOL;
T_High_oil_filter_diff_press : BOOL;
T_Flow_switch_FT01 : BOOL;
T_Starter_failure_trip : BOOL;
T_Incorrect_feedback_starter_trip : BOOL;


A_High_condenser_flow : BOOL;
A_Rotating_stall : BOOL;
A_High_temp_oil_inlet_comp : BOOL;
SpareAlarm_1 : BOOL;
A_High_motor_air_temp : BOOL;
A_High_control_panel_temp : BOOL;
A_Low_oil_diff_pressure : BOOL;
Spare_alarm_2 : BOOL;
A_High_comp_motor_winding_temp : BOOL;
A_High_comp_mo_DE_bear_temp : BOOL;
A_High_comp_mo_NDE_bear_temp : BOOL;
A_High_comp_mo_DE_bear_vib : BOOL;
A_High_comp_mo_NDE_bear_vib : BOOL;
A_Low_chilled_medium_flow : BOOL;
A_High_chilled_medium_flow : BOOL;
A_Low_sea_water_flow : BOOL;
A_Seawater_pump_not_running : BOOL;
A_Spare : BOOL;
A_Spare_1 : BOOL;
A_Spare_2 : BOOL;
A_Spare_3 : BOOL;
A_Spare_4 : BOOL;
A_Spare_5 : BOOL;
A_Spare_6 : BOOL;
A_Spare_7 : BOOL;
A_Spare_8 : BOOL;
A_Spare_9 : BOOL;
A_Spare_10 : BOOL;
A_Spare_11 : BOOL;
A_High_oil_filter_diff_press : BOOL;
A_Spare_12 : BOOL;
A_Spare_13 : BOOL;
A_Spare_14 : BOOL;
A_Spare_15 : BOOL;
A_Spare_16 : BOOL;
A_Spare_17 : BOOL;
Anti_recycle_status : BOOL;
Low_oil_temperature : BOOL;
Low_oil_temp_auto : BOOL;
Oil_heater : BOOL;
Sea_water_pump : BOOL;
Comp_oil_pump : BOOL;
Bearing_oil_pump : BOOL;
Solenoid_oil_return : BOOL;
Unit_running : BOOL;
Unit_remote : BOOL;
Unit_auto : BOOL;
Unit_manual : BOOL;
Unit_trip : BOOL;
Unit_alarm : BOOL;
Unit_start_switch : BOOL;
Unit_available : BOOL;
S_Spare_1 : BOOL;
S_Spare_2 : BOOL;
S_Spare_3 : BOOL;
S_Spare_4 : BOOL;
S_Spare_5 : BOOL;
S_Spare_6 : BOOL;
S_Spare_7 : BOOL;
S_Spare_8 : BOOL;
Solenoid_liquid_inj: BOOL;
CW_Flow_ind : BOOL;
Open_chilled_water_valve : BOOL;
Feedback_chilled_water_valve : BOOL;
Open_order_swv_overboard : BOOL;
Close_order_swv_overboard : BOOL;
Open_order_swv_bypass : BOOL;
Close_order_swv_bypass : BOOL;
VFD_man_auto : BOOL ;
VFD_freq_jump_on : BOOL ;
VFD_ramp_100_perc : BOOL ;
VFD_locked_100_perc : BOOL;
VFD_ramp_d_PRVcontrol : BOOL;
PRV_control : BOOL;
VFD_control : BOOL;
VFD_fixed_speed : BOOL;
Spare_151: BOOL;
T_Transformer_winding_temp : BOOL;
A_Transformer_winding_temp : BOOL;
T_trafo_opening_main_breaker : BOOL;
T_VFD : BOOL;
VFD_ready : BOOL;
T_VFD_emergency_stop : BOOL;
T_Low_5VDC_supply : BOOL;
T_High_5VDC_supply : BOOL;
T_Spare_9 : BOOL;
T_Spare_10 : BOOL;
T_Spare_11 : BOOL;
T_Spare_12 : BOOL;
T_Spare_13 : BOOL;
T_Low_liquid_level : BOOL;
T_SW_pump_off_to_long : BOOL;
T_Softstarter_failure : BOOL;
T_Motorstarter_failure : BOOL ;
T_CW_valveopen_failure : BOOL ;
T_SW_valveopen_failure : BOOL ;
T_High_disch_superheat :BOOL ;
T_Low_disch_superheat :BOOL ;
T_High_CW_outlet_temp : BOOL;
T_Low_CW_outlet_temp : BOOL;
T_Low_CW_inlet_temp : BOOL;
T_High_CW_inlet_temp : BOOL;
T_High_SW_outlet_temp : BOOL;
T_Low_SW_outlet_temp : BOOL;
T_Low_SW_inlet_temp : BOOL;
T_High_SW_inlet_temp : BOOL;
T_High_motor_wind_temp_R : BOOL;
T_High_motor_wind_temp_S : BOOL;
T_High_motor_wind_temp_T : BOOL;
T_High_press_ratio : BOOL;
T_Low_press_ratio : BOOL;
T_Low_CW_dP : BOOL;
T_High_CW_dP : BOOL;
T_Low_SW_dP : BOOL;
T_High_SW_dP : BOOL;
T_Long_time_PRV : BOOL;
T_Comp_thrust_neg_move : BOOL;
T_Comp_thrust_pos_move : BOOL;
T_VGD_fault : BOOL;
T_Low_oilpress_prelube : BOOL;
T_Low_temp_oil_inlet_comp : BOOL;
T_Low_oilpress_standby : BOOL;
T_Transformer : BOOL;
A_Transformer : BOOL;


T_Sensor_low_signal_AI_64 : BOOL;
T_Sensor_high_signal_AI_64 : BOOL;
T_Sensor_low_signal_AI_66 : BOOL;
T_Sensor_high_signal_AI_66 : BOOL;
T_Sensor_low_signal_AI_112 : BOOL;
T_Sensor_high_signal_AI_112 : BOOL;
T_Sensor_low_signal_AI_114 : BOOL;
T_Sensor_high_signal_AI_114 : BOOL;
T_Sensor_low_signal_AI_116 : BOOL;
T_Sensor_high_signal_AI_116 : BOOL;
T_Sensor_low_signal_AI_118 : BOOL;
T_Sensor_high_signal_AI_118 : BOOL;
T_Sensor_high_signal_AI_128 : BOOL;
T_Sensor_low_signal_AI_128 : BOOL ;
T_Sensor_high_signal_AI_130 : BOOL;
T_Sensor_low_signal_AI_130 : BOOL ;
T_Sensor_high_signal_AI_132 : BOOL;
T_Sensor_low_signal_AI_132 : BOOL ;
T_Sensor_high_signal_AI_134 : BOOL;
T_Sensor_low_signal_AI_134 : BOOL ;
T_Sensor_high_signal_AI_136 : BOOL;
T_Sensor_low_signal_AI_136 : BOOL ;
T_Sensor_high_signal_AI_138 : BOOL;
T_Sensor_low_signal_AI_138 : BOOL ;
T_Sensor_high_signal_AI_140 : BOOL;
T_Sensor_low_signal_AI_140 : BOOL ;
T_Sensor_high_signal_AI_142 : BOOL;
T_Sensor_low_signal_AI_142 : BOOL ;
T_Sensor_high_signal_AI_144 : BOOL;
T_Sensor_low_signal_AI_144 : BOOL ;
T_Sensor_high_signal_AI_146 : BOOL;
T_Sensor_low_signal_AI_146 : BOOL ;
T_Sensor_high_signal_AI_148 : BOOL;
T_Sensor_low_signal_AI_148 : BOOL ;
T_Sensor_high_signal_AI_150 : BOOL;
T_Sensor_low_signal_AI_150 : BOOL ;
T_Sensor_high_signal_AI_152 : BOOL;
T_Sensor_low_signal_AI_152 : BOOL ;
T_Sensor_high_signal_AI_154 : BOOL;
T_Sensor_low_signal_AI_154 : BOOL ;
T_Sensor_high_signal_AI_156 : BOOL;
T_Sensor_low_signal_AI_156 : BOOL ;
T_Sensor_high_signal_AI_158 : BOOL;
T_Sensor_low_signal_AI_158 : BOOL ;
T_Sensor_high_signal_AI_160 : BOOL;
T_Sensor_low_signal_AI_160 : BOOL ;
T_Sensor_high_signal_AI_162 : BOOL;
T_Sensor_low_signal_AI_162 : BOOL ;
T_Sensor_high_signal_AI_164 : BOOL;
T_Sensor_low_signal_AI_164 : BOOL ;
T_Sensor_high_signal_AI_166 : BOOL;
T_Sensor_low_signal_AI_166 : BOOL ;
T_Sensor_high_signal_AI_168 : BOOL;
T_Sensor_low_signal_AI_168 : BOOL ;
T_Sensor_high_signal_AI_170 : BOOL;
T_Sensor_low_signal_AI_170 : BOOL ;
T_Sensor_high_signal_AI_172 : BOOL;
T_Sensor_low_signal_AI_172 : BOOL ;
T_Sensor_high_signal_AI_174 : BOOL;
T_Sensor_low_signal_AI_174 : BOOL ;
T_Sensor_high_signal_AI_176 : BOOL;
T_Sensor_low_signal_AI_176 : BOOL ;
T_Sensor_low_signal_AI_178 : BOOL ;
T_Sensor_high_signal_AI_178 : BOOL;
T_Sensor_low_signal_AI_180 : BOOL ;
T_Sensor_high_signal_AI_180 : BOOL;
T_Sensor_low_signal_AI_182 : BOOL ;
T_Sensor_high_signal_AI_182 : BOOL;
T_Sensor_low_signal_AI_184 : BOOL ;
T_Sensor_high_signal_AI_184 : BOOL;
T_Sensor_low_signal_AI_186 : BOOL ;
T_Sensor_high_signal_AI_186 : BOOL;
T_Sensor_low_signal_AI_188 : BOOL ;
T_Sensor_high_signal_AI_188 : BOOL;
T_Sensor_low_signal_AI_190 : BOOL ;
T_Sensor_high_signal_AI_190 : BOOL;
T_Sensor_low_signal_AI_192 : BOOL ;
T_Sensor_high_signal_AI_192 : BOOL;
T_Sensor_low_signal_AI_194 : BOOL ;
T_Sensor_high_signal_AI_194 : BOOL;
T_Sensor_low_signal_AI_196 : BOOL ;
T_Sensor_high_signal_AI_196 : BOOL;
T_Sensor_low_signal_AI_198 : BOOL ;
T_Sensor_high_signal_AI_198 : BOOL;
T_Sensor_high_signal_AI_200 : BOOL;
T_Sensor_low_signal_AI_200 : BOOL ;
T_Sensor_low_signal_AI_202 : BOOL ;
T_Sensor_high_signal_AI_202 : BOOL;
T_Sensor_low_signal_AI_204 : BOOL ;
T_Sensor_high_signal_AI_204 : BOOL;
T_Sensor_low_signal_AI_206 : BOOL ;
T_Sensor_high_signal_AI_206 : BOOL ;
CW_Pump_Remote_Start_Available : BOOL;
T_CW_Pump : BOOL;
A_high_disch_press : BOOL ;
A_low_disch_press : BOOL ;
A_Low_suction_pressure : BOOL;
A_High_suction_pressure : BOOL;
A_High_discharge_temp : BOOL;
A_High_oil_temp_receiver : BOOL;
A_Low_oil_temp_receiver : BOOL;
A_Low_temp_oil_inlet_comp : BOOL;
A_High_oil_diff_pressure : BOOL;
A_Low_discharge_superheat : BOOL;
A_High_discharge_superheat : BOOL;
A_Low_CW_outlet_temp : BOOL;
A_High_CW_outlet_temp : BOOL;
A_Low_CW_inlet_temp : BOOL;
A_High_CW_inlet_temp : BOOL;
A_High_SW_outlet_temp : BOOL;
A_Low_condenser_flow : BOOL;
A_High_press_ratio : BOOL;
A_Low_press_ratio : BOOL;
A_Motor_speed_low : BOOL;
A_Low_SW_outlet_temp : BOOL;
A_Low_SW_inlet_temp : BOOL;
A_High_SW_inlet_temp : BOOL;
A_High_suction_superheat : BOOL;
A_Low_suction_superheat : BOOL;
A_High_temp_oil_separator : BOOL;
A_Low_temp_oil_separator : BOOL;
A_High_motor_wind_temp_R : BOOL;
A_High_motor_wind_temp_S : BOOL;
A_High_motor_wind_temp_T : BOOL;
A_High_CW_dP : BOOL;
A_Low_CW_dP : BOOL;
A_High_SW_dP : BOOL;
A_Low_SW_dP : BOOL;
A_VGD_Fault : BOOL;
Start_inhib_time_between_Start : BOOL;
Start_inhib_time_between_Stop_Start : BOOL;
Start_inhib_PRV_not_min : BOOL;
Start_inhib_Motor_overload : BOOL;
Remote_bilge_pump_control : BOOL;
CW_pump_running : BOOL;
A_Low_liquid_level : BOOL;
A_Suction_press_limit : BOOL;
A_Discharge_press_limit : BOOL;
A_Discharge_superheat_limit : BOOL;
A_Motor_current_limit : BOOL;


DI_0_0_Emergency_stop : BOOL;
DI_0_1 : BOOL;
DI_0_2_Fault_reset : BOOL;
DI_0_3 : BOOL;
DI_0_4 : BOOL;
DI_0_5 : BOOL;
DI_0_6_Overload_protection : BOOL;
DI_0_7 : BOOL;
DI_1_0_Overload_oilpump : BOOL;
DI_1_1 : BOOL;
DI_1_2 : BOOL;
DI_1_3 : BOOL;
DI_1_4_Power_available : BOOL;
DI_1_5_Starter_failure : BOOL;
DI_8_0_Controlpanel_temp : BOOL;
DI_8_1 : BOOL;
DI_8_2_VGD_limit_switch : BOOL;
DI_8_3_water_leak_motor  : BOOL;
DI_8_4_Catodic_protection : BOOL;
DI_8_5_Trust_bearing_probe : BOOL;
DI_8_6_ESD_operation : BOOL;
DI_8_7 : BOOL;
DI_9_0_MV_breaker_available : BOOL;
DI_9_1 : BOOL;
DI_9_2_Safe_return_to_port : BOOL;
DI_9_3 : BOOL;
DI_9_4_VFD_emergency_stop : BOOL;
DI_9_5 : BOOL;
DI_9_6 : BOOL;
DI_9_7 : BOOL;
DO_0_0_Start_signal_comp : BOOL;
DO_0_1_Start_signal_oil_pump : BOOL;
DO_0_2_Start_signal_SW_pump : BOOL;
DO_0_3_Start_signal_CW_pump : BOOL;
DO_0_4_Solenoid_valve_oil : BOOL;
DO_0_5_Solenoid_valve_liquid : BOOL;
DO_0_6_Oil_heater : BOOL;
DO_0_7_Comp_heater : BOOL;
DO_1_0 : BOOL;
DO_1_1 : BOOL;
DO_8_0_Liquid_valve_open : BOOL;
DO_8_1_Liquid_valve_close : BOOL;
DO_8_2_VGD_open : BOOL;
DO_8_3_VGD_close : BOOL;
DO_8_4_PRV_open : BOOL;
DO_8_5_PRV_close : BOOL;
DO_8_6_HGV_open : BOOL;
DO_8_7_HGV_close : BOOL;
DO_9_0_Main_breaker_ready : BOOL;
DO_9_1_Close_order_swv_overboard : BOOL;
DO_9_2_Open_order_swv_bypass : BOOL;
DO_9_3_Close_order_swv_bypass : BOOL;
DO_9_4 : BOOL;
DO_9_5 : BOOL;
DO_9_6 : BOOL;
DO_9_7 : BOOL;
DO_12_0_Power_request : BOOL;
DO_12_1_Compressor_ready : BOOL;
DO_12_2 : BOOL;
DO_12_3 : BOOL;
DO_12_4_Control_panel_alarm : BOOL;
DO_12_5_Auto_reset : BOOL;
DO_12_6_Unit_running : BOOL;
DO_12_7_Emergency_MV_Breaker : BOOL;
Start_inhib_time_Oil_receiver_temp : BOOL;



//Graphic variables
Unit_switch_status : INT;
i : INT;
show_trendvalue : ARRAY[0..50] OF BOOL;
select_trendvalue : INT :=0 ;

END_VAR

modbus_var[0] :=%IW0;
Temp_discharge:=wordstoReal(modbus_var_1000[1],modbus_var_1000[0]);
Liquid_line_temp:=wordstoReal(modbus_var_1000[3],modbus_var_1000[2]);
Oil_temp_receiver:=wordstoReal(modbus_var_1000[5],modbus_var_1000[4]);
Temp_oil_inlet_compr:=wordstoReal(modbus_var_1000[7],modbus_var_1000[6]);
Temp_water_inlet_cond:=wordstoReal(modbus_var_1000[9],modbus_var_1000[8]);
Temp_water_outlet_cond:=wordstoReal(modbus_var_1000[11],modbus_var_1000[10]);
Temp_chilled_medium_in:=wordstoReal(modbus_var_1000[13],modbus_var_1000[12]);
Temp_chilled_medium_out:=wordstoReal(modbus_var_1000[15],modbus_var_1000[14]);
Temp_motor_wind_R:=wordstoReal(modbus_var_1000[17],modbus_var_1000[16]);
Temp_motor_wind_S:=wordstoReal(modbus_var_1000[19],modbus_var_1000[18]);
Temp_motor_wind_T:=wordstoReal(modbus_var_1000[21],modbus_var_1000[20]);
Temp_motor_bearing_DE:=wordstoReal(modbus_var_1000[23],modbus_var_1000[22]);
Temp_motor_bearing_NDE:=wordstoReal(modbus_var_1000[25],modbus_var_1000[24]);
Temp_motor_air:=wordstoReal(modbus_var_1000[27],modbus_var_1000[26]);
Spare:=wordstoReal(modbus_var_1000[29],modbus_var_1000[28]);
Spare:=wordstoReal(modbus_var_1000[31],modbus_var_1000[30]);
Spare:=wordstoReal(modbus_var_1000[33],modbus_var_1000[32]);
Spare:=wordstoReal(modbus_var_1000[35],modbus_var_1000[34]);
Spare:=wordstoReal(modbus_var_1000[37],modbus_var_1000[36]);
Spare:=wordstoReal(modbus_var_1000[39],modbus_var_1000[38]);
Spare:=wordstoReal(modbus_var_1000[41],modbus_var_1000[40]);
Spare:=wordstoReal(modbus_var_1000[43],modbus_var_1000[42]);
Spare:=wordstoReal(modbus_var_1000[45],modbus_var_1000[44]);
Spare:=wordstoReal(modbus_var_1000[47],modbus_var_1000[46]);
Press_discharge_compr:=wordstoReal(modbus_var_1000[49],modbus_var_1000[48]);
Press_suction_compr:=wordstoReal(modbus_var_1000[51],modbus_var_1000[50]);
Press_oil_receiver:=wordstoReal(modbus_var_1000[53],modbus_var_1000[52]);
Oil_pressure_before_filter:=wordstoReal(modbus_var_1000[55],modbus_var_1000[54]);
Press_oil_compr:=wordstoReal(modbus_var_1000[57],modbus_var_1000[56]);
Press_water_cond_inlet:=wordstoReal(modbus_var_1000[59],modbus_var_1000[58]);
Press_water_cond_out:=wordstoReal(modbus_var_1000[61],modbus_var_1000[60]);
Spare:=wordstoReal(modbus_var_1000[63],modbus_var_1000[62]);
Press_chilled_medium_in:=wordstoReal(modbus_var_1000[65],modbus_var_1000[64]);
Press_chilled_medium_out:=wordstoReal(modbus_var_1000[67],modbus_var_1000[66]);
Motor_current:=wordstoReal(modbus_var_1000[69],modbus_var_1000[68]);
Speed_feedback_VFD:=wordstoReal(modbus_var_1000[71],modbus_var_1000[70]);
Vibration_compressor_DE:=wordstoReal(modbus_var_1000[73],modbus_var_1000[72]);
Vibration_compressor_NDE:=wordstoReal(modbus_var_1000[75],modbus_var_1000[74]);
VFD_motor_current:=wordstoReal(modbus_var_1000[77],modbus_var_1000[76]);
Spare:=wordstoReal(modbus_var_1000[79],modbus_var_1000[78]);
Feedback_liquid_valve_raw:=wordstoReal(modbus_var_1000[81],modbus_var_1000[80]);
Feedback_VGD_raw:=wordstoReal(modbus_var_1000[83],modbus_var_1000[82]);
Feedback_PRV_raw:=wordstoReal(modbus_var_1000[85],modbus_var_1000[84]);
Feedback_HGV_raw:=wordstoReal(modbus_var_1000[87],modbus_var_1000[86]);
Feedback_seawater_valve_overboard_raw:=wordstoReal(modbus_var_1000[89],modbus_var_1000[88]); 
Feedback_seawater_valve_bypass_raw:=wordstoReal(modbus_var_1000[91],modbus_var_1000[90]);
Thrust_bearing_position:=wordstoReal(modbus_var_1000[93],modbus_var_1000[92]);
Spare:=wordstoReal(modbus_var_1000[95],modbus_var_1000[94]);
Stall_detector:=wordstoReal(modbus_var_1000[97],modbus_var_1000[96]);
Liquid_level_condenser:=wordstoReal(modbus_var_1000[99],modbus_var_1000[98]);
Spare:=wordstoReal(modbus_var_1000[101],modbus_var_1000[100]);
Spare:=wordstoReal(modbus_var_1000[103],modbus_var_1000[102]);
Spare:=wordstoReal(modbus_var_1000[105],modbus_var_1000[104]);
Spare:=wordstoReal(modbus_var_1000[107],modbus_var_1000[106]);
Spare:=wordstoReal(modbus_var_1000[109],modbus_var_1000[108]);
Spare:=wordstoReal(modbus_var_1000[111],modbus_var_1000[110]);
Spare:=wordstoReal(modbus_var_1000[113],modbus_var_1000[112]);
Spare:=wordstoReal(modbus_var_1000[115],modbus_var_1000[114]);
Chiller_capacity_kW:=wordstoReal(modbus_var_1000[117],modbus_var_1000[116]);
Chiller_capacity_t1:=wordstoReal(modbus_var_1000[119],modbus_var_1000[118]);
Chiller_capacity:=wordstoReal(modbus_var_1000[121],modbus_var_1000[120]);
Control_signal_unit_d:=wordstoReal(modbus_var_1000[123],modbus_var_1000[122]);

COP_chiller_mech:=wordstoReal(modbus_var_1001[125],modbus_var_1001[124]);
Spare:=wordstoReal(modbus_var_1001[127],modbus_var_1001[126]);
Spare:=wordstoReal(modbus_var_1001[129],modbus_var_1001[128]);
Spare:=wordstoReal(modbus_var_1001[131],modbus_var_1001[130]);
Spare:=wordstoReal(modbus_var_1001[133],modbus_var_1001[132]);
P2_mot_1_kW:=wordstoReal(modbus_var_1001[135],modbus_var_1001[134]);
SP_MC_controller:=wordstoReal(modbus_var_1001[137],modbus_var_1001[136]);
Max_motor_wind_temp:=wordstoReal(modbus_var_1001[139],modbus_var_1001[138]);
Running_hours_compressormotor:=wordstoReal(modbus_var_1001[141],modbus_var_1001[140]);
Spare:=wordstoReal(modbus_var_1001[143],modbus_var_1001[142]);
Spare:=wordstoReal(modbus_var_1001[145],modbus_var_1001[144]);
Spare:=wordstoReal(modbus_var_1001[147],modbus_var_1001[146]);
Spare:=wordstoReal(modbus_var_1001[149],modbus_var_1001[148]);
Discharge_saturated_temp:=wordstoReal(modbus_var_1001[151],modbus_var_1001[150]);
SP_cond_press:=wordstoReal(modbus_var_1001[153],modbus_var_1001[152]);
SP_cond_press_limit:=wordstoReal(modbus_var_1001[155],modbus_var_1001[154]);    // Double defined?
Discharge_superheat:=wordstoReal(modbus_var_1001[157],modbus_var_1001[156]); 
SP_discharge_superheat_limit:=wordstoReal(modbus_var_1001[159],modbus_var_1001[158]);
SP_PID_Level:=wordstoReal(modbus_var_1001[161],modbus_var_1001[160]);
Liquid_valve_output:=wordstoReal(modbus_var_1001[163],modbus_var_1001[162]);    // Sequence control signal
Feedback_liquid_valve:=wordstoReal(modbus_var_1001[165],modbus_var_1001[164]); 
dP_SW:=wordstoReal(modbus_var_1001[167],modbus_var_1001[166]);
SW_pump_speed_order:=wordstoReal(modbus_var_1001[169],modbus_var_1001[168]);
Order_SWW_overboard:=wordstoReal(modbus_var_1001[171],modbus_var_1001[170]);
Order_SWW_bypass:=wordstoReal(modbus_var_1001[173],modbus_var_1001[172]);
Feedback_seawater_valve_overboard:=wordstoReal(modbus_var_1001[175],modbus_var_1001[174]);
Feedback_seawater_valve_bypass:=wordstoReal(modbus_var_1001[177],modbus_var_1001[176]);
Spare:=wordstoReal(modbus_var_1001[179],modbus_var_1001[178]);
Spare:=wordstoReal(modbus_var_1001[181],modbus_var_1001[180]);
Spare:=wordstoReal(modbus_var_1001[183],modbus_var_1001[182]);
Spare:=wordstoReal(modbus_var_1001[185],modbus_var_1001[184]);
SP_CW_controller:=wordstoReal(modbus_var_1001[187],modbus_var_1001[186]);
Suction_saturated_temp:=wordstoReal(modbus_var_1001[189],modbus_var_1001[188]);
SP_evap_press_limit:=wordstoReal(modbus_var_1001[191],modbus_var_1001[190]);
Theta_out:=wordstoReal(modbus_var_1001[193],modbus_var_1001[192]);
dP_CW:=wordstoReal(modbus_var_1001[195],modbus_var_1001[194]);
Spare:=wordstoReal(modbus_var_1001[197],modbus_var_1001[196]);
Spare:=wordstoReal(modbus_var_1001[199],modbus_var_1001[198]);
Spare:=wordstoReal(modbus_var_1001[201],modbus_var_1001[200]);
Spare:=wordstoReal(modbus_var_1001[203],modbus_var_1001[202]);
SP_oil_pressure:=wordstoReal(modbus_var_1001[205],modbus_var_1001[204]);
Oil_diff_pressure:=wordstoReal(modbus_var_1001[207],modbus_var_1001[206]);
Oil_Filter_Drop:=wordstoReal(modbus_var_1001[209],modbus_var_1001[208]);
Setpoint_conv_oil_pump:=wordstoReal(modbus_var_1001[211],modbus_var_1001[210]);
Oil_pump_running_hours:=wordstoReal(modbus_var_1001[213],modbus_var_1001[212]);
Spare:=wordstoReal(modbus_var_1001[215],modbus_var_1001[214]);
Spare:=wordstoReal(modbus_var_1001[217],modbus_var_1001[216]);
Spare:=wordstoReal(modbus_var_1001[219],modbus_var_1001[218]);
Spare:=wordstoReal(modbus_var_1001[221],modbus_var_1001[220]);
Thrust_bearing_ref:=wordstoReal(modbus_var_1001[223],modbus_var_1001[222]);
Prerotary_output:=wordstoReal(modbus_var_1001[225],modbus_var_1001[224]);
Feedback_PRV:=wordstoReal(modbus_var_1001[227],modbus_var_1001[226]);
Min_allowed_PRVposition:=wordstoReal(modbus_var_1001[229],modbus_var_1001[228]);
VGD_output:=wordstoReal(modbus_var_1001[231],modbus_var_1001[230]);
Feedback_VGD:=wordstoReal(modbus_var_1001[233],modbus_var_1001[232]);
Stall_ramp:=wordstoReal(modbus_var_1001[235],modbus_var_1001[234]);
Hot_gas_valve_output:=wordstoReal(modbus_var_1001[237],modbus_var_1001[236]);
Feedback_HGV:=wordstoReal(modbus_var_1001[239],modbus_var_1001[238]);
Spare:=wordstoReal(modbus_var_1001[241],modbus_var_1001[240]);
Spare:=wordstoReal(modbus_var_1001[243],modbus_var_1001[242]);
Spare:=wordstoReal(modbus_var_1001[245],modbus_var_1001[244]);
Spare:=wordstoReal(modbus_var_1001[247],modbus_var_1001[246]);

Opt_speed_VFD_perc:=wordstoReal(modbus_var_1002[249],modbus_var_1002[248]);
Order_VFD_Hz:=wordstoReal(modbus_var_1002[251],modbus_var_1002[250]);
Speed_feedback_VFD:=wordstoReal(modbus_var_1002[253],modbus_var_1002[252]);
VFD_min_allowed_frequence:=wordstoReal(modbus_var_1002[255],modbus_var_1002[254]);
VFD_min_allowed_speed:=wordstoReal(modbus_var_1002[257],modbus_var_1002[256]);
Spare:=wordstoReal(modbus_var_1002[259],modbus_var_1002[258]);
CW_Pump_Speed_SP:=wordstoReal(modbus_var_1002[261],modbus_var_1002[260]);
Spare:=wordstoReal(modbus_var_1002[263],modbus_var_1002[262]);
Spare:=wordstoReal(modbus_var_1002[265],modbus_var_1002[264]);
Spare:=wordstoReal(modbus_var_1002[267],modbus_var_1002[266]);
Spare:=wordstoReal(modbus_var_1002[269],modbus_var_1002[268]);
Spare:=wordstoReal(modbus_var_1002[271],modbus_var_1002[270]);
Spare:=wordstoReal(modbus_var_1002[273],modbus_var_1002[272]);
Spare:=wordstoReal(modbus_var_1002[275],modbus_var_1002[274]);
//PI_chiller_write:=wordstoReal(modbus_var_1002[277],modbus_var_1002[276]);
//Wasted_energy_kW_write:=wordstoReal(modbus_var_1002[279],modbus_var_1002[278]);
Spare:=wordstoReal(modbus_var_1002[281],modbus_var_1002[280]);
P1_motor_kW:=wordstoReal(modbus_var_1002[283],modbus_var_1002[282]);
COP_chiller_ele:=wordstoReal(modbus_var_1002[285],modbus_var_1002[284]);
//PI_chiller:=wordstoReal(modbus_var_1002[287],modbus_var_1002[286]);
//Wasted_energy_kW:=wordstoReal(modbus_var_1002[289],modbus_var_1002[288]);
Cal_date_MMYY:=wordstoReal(modbus_var_1002[291],modbus_var_1002[290]);
Spare:=wordstoReal(modbus_var_1002[293],modbus_var_1002[292]);
Spare:=wordstoReal(modbus_var_1002[295],modbus_var_1002[294]);
Spare:=wordstoReal(modbus_var_1002[297],modbus_var_1002[296]);

// Write PI to PLC
modbus_var_1002[276]:=modbusslave_com.sequence_lowByte_PI_ch_5;
modbus_var_1002[277]:=modbusslave_com.sequence_highByte_PI_ch_5;
modbus_var_1002[278]:=modbusslave_com.sequence_lowByte_Wasted_energy_ch_5_kW;
modbus_var_1002[279]:=modbusslave_com.sequence_highByte_Wasted_energy_ch_5_kW;

// Word variables
Anti_recycle_time:=scaleFunction(modbus_var_1002[300],1.0, 0);
Number_of_starts:=scaleFunction(modbus_var_1002[301],1.0, 0);
Q2_chillerMWh:=scaleFunction(modbus_var_1002[302],1.0, 0);
Chiller_P1_MWh:=scaleFunction(modbus_var_1002[303],1.0, 0);
Alarm_limit_stall_count:=scaleFunction(modbus_var_1002[304],1.0, 0);
Days_above_stall_limit:=scaleFunction(modbus_var_1002[305],1.0, 0);
Hrs_above_stall_limit:=scaleFunction(modbus_var_1002[306],1.0, 0);
Min_above_stall_limit:=scaleFunction(modbus_var_1002[307],1.0, 0);
Sec_above_stall_limit:=scaleFunction(modbus_var_1002[308],1.0, 0);
Surge_counter_VFD:=scaleFunction(modbus_var_1002[309],1.0, 0);

Trip_BITs_0_to_15:=modbus_var_1002[340];
Trip_BITs_16_to_31:=modbus_var_1002[341];
Trip_BITs_32_to_47:=modbus_var_1002[342];
Trip_BITs_48_to_63:=modbus_var_1002[343];
Trip_BITs_64_to_79:=modbus_var_1002[344];
Trip_BITs_80_to_95:=modbus_var_1002[345];
Trip_BITs_96_to_121:=modbus_var_1002[346];
Trip_BITs_122_to_137:=modbus_var_1002[347];
Trip_BITs_138_to_153:=modbus_var_1002[348];
Trip_BITs_154_to_169:=modbus_var_1002[349];
Trip_BITs_170_to_185:=modbus_var_1002[350];
Trip_BITs_186_to_201:=modbus_var_1002[351];

Alarm_BITs_0_to_15:=modbus_var_1002[360];
Alarm_BITs_16_to_31:=modbus_var_1002[361];
Alarm_BITs_32_to_47:=modbus_var_1002[362];
Alarm_BITs_48_to_63:=modbus_var_1002[363];
Alarm_BITs_64_to_79:=modbus_var_1002[364];

Status_BITs_0_to_15:=modbus_var_1002[330];
Status_BITs_16_to_31:=modbus_var_1002[331];
Status_BITs_32_to_47:=modbus_var_1002[332];
Status_BITs_48_to_63:=modbus_var_1002[333];
Status_BITs_64_to_79:=modbus_var_1002[334];
Status_BITs_80_to_95:=modbus_var_1002[335];


// Trip bits
T_Low_discharge_pressure:=maskbitFunction(Trip_BITs_0_to_15,0);
T_High_discharge_pressure:=maskbitFunction(Trip_BITs_0_to_15,1);
T_Low_suction_pressure:=maskbitFunction(Trip_BITs_0_to_15,2);
T_High_suction_pressure:=maskbitFunction(Trip_BITs_0_to_15,3);
T_Low_press_ratio:=maskbitFunction(Trip_BITs_0_to_15,4);
T_High_discharge_temp:=maskbitFunction(Trip_BITs_0_to_15,5);
T_Low_disch_superheat:=maskbitFunction(Trip_BITs_0_to_15,6);
T_High_disch_superheat:=maskbitFunction(Trip_BITs_0_to_15,7);
S_Spare_1:=maskbitFunction(Trip_BITs_0_to_15,8);
S_Spare_1:=maskbitFunction(Trip_BITs_0_to_15,9);
T_Low_temp_oil_inlet_comp:=maskbitFunction(Trip_BITs_0_to_15,10);
T_High_temp_oil_inlet_comp:=maskbitFunction(Trip_BITs_0_to_15,11);
T_Low_temp_oil_receiver:=maskbitFunction(Trip_BITs_0_to_15,12);
T_High_temp_oil_receiver:=maskbitFunction(Trip_BITs_0_to_15,13);
T_Low_oil_diff_pressure:=maskbitFunction(Trip_BITs_0_to_15,14);
T_High_diff_oil_pressure:=maskbitFunction(Trip_BITs_0_to_15,15);
T_Low_oilpress_prelube:=maskbitFunction(Trip_BITs_16_to_31,0);

T_Low_oilpress_standby:=maskbitFunction(Trip_BITs_16_to_31,1);
T_High_oil_filter_diff_press:=maskbitFunction(Trip_BITs_16_to_31,2);
T_Oil_pump_running_failure:=maskbitFunction(Trip_BITs_16_to_31,3);
T_Overload_oil_pump_motor:=maskbitFunction(Trip_BITs_16_to_31,4);
S_Spare_1:=maskbitFunction(Trip_BITs_16_to_31,5);
S_Spare_1:=maskbitFunction(Trip_BITs_16_to_31,6);
T_Low_CW_outlet_temp:=maskbitFunction(Trip_BITs_16_to_31,7);
T_High_CW_inlet_temp:=maskbitFunction(Trip_BITs_16_to_31,8);
T_Low_CW_dP:=maskbitFunction(Trip_BITs_16_to_31,9);
T_High_CW_dP:=maskbitFunction(Trip_BITs_16_to_31,10);
T_Flow_switch_FT01:=maskbitFunction(Trip_BITs_16_to_31,11);
T_Chilled_pump_run_failure:=maskbitFunction(Trip_BITs_16_to_31,12);
T_CW_valveopen_failure:=maskbitFunction(Trip_BITs_16_to_31,13);
S_Spare_1:=maskbitFunction(Trip_BITs_16_to_31,14);
S_Spare_1:=maskbitFunction(Trip_BITs_16_to_31,15);

T_Low_SW_inlet_temp:=maskbitFunction(Trip_BITs_32_to_47,0);
T_High_SW_inlet_temp:=maskbitFunction(Trip_BITs_32_to_47,1);
T_Low_SW_dP:=maskbitFunction(Trip_BITs_32_to_47,2);
T_High_SW_dP:=maskbitFunction(Trip_BITs_32_to_47,3);
T_Sea_water_pump_run_failure:=maskbitFunction(Trip_BITs_32_to_47,4);
T_SW_valveopen_failure:=maskbitFunction(Trip_BITs_32_to_47,5);
T_Low_liquid_level:=maskbitFunction(Trip_BITs_32_to_47,6);
T_Cathodic_protect_sys_alarm:=maskbitFunction(Trip_BITs_32_to_47,7);
S_Spare_1:=maskbitFunction(Trip_BITs_32_to_47,8);
S_Spare_1:=maskbitFunction(Trip_BITs_32_to_47,9);
T_High_motor_wind_temp_R:=maskbitFunction(Trip_BITs_32_to_47,10);
T_High_motor_wind_temp_S:=maskbitFunction(Trip_BITs_32_to_47,11);
T_High_motor_wind_temp_T:=maskbitFunction(Trip_BITs_32_to_47,12);
T_High_comp_mot_DE_bear_temp:=maskbitFunction(Trip_BITs_32_to_47,13);
T_High_comp_mot_NDE_bear_temp:=maskbitFunction(Trip_BITs_32_to_47,14);
T_High_motor_air_temp:=maskbitFunction(Trip_BITs_32_to_47,15);

T_High_comp_mot_DE_bear_vib:=maskbitFunction(Trip_BITs_48_to_63,0);
T_High_comp_mot_NDE_bear_vib:=maskbitFunction(Trip_BITs_48_to_63,1);
T_Comp_motor_leak_detection:=maskbitFunction(Trip_BITs_48_to_63,2);
T_Comp_motor_power_loss:=maskbitFunction(Trip_BITs_48_to_63,3);
T_Starter_failure_trip:=maskbitFunction(Trip_BITs_48_to_63,4);
T_Overload_compressor_motor:=maskbitFunction(Trip_BITs_48_to_63,5);
T_Compressor_running_failure:=maskbitFunction(Trip_BITs_48_to_63,6);
T_Incorrect_feedback_starter_trip:=maskbitFunction(Trip_BITs_48_to_63,7);
T_Softstarter_failure:=maskbitFunction(Trip_BITs_48_to_63,8);
T_VFD:=maskbitFunction(Trip_BITs_48_to_63,9);
T_Emergency_stop:=maskbitFunction(Trip_BITs_48_to_63,10);
S_Spare_1:=maskbitFunction(Trip_BITs_48_to_63,11);
S_Spare_1:=maskbitFunction(Trip_BITs_48_to_63,12);
S_Spare_1:=maskbitFunction(Trip_BITs_48_to_63,13);
S_Spare_1:=maskbitFunction(Trip_BITs_48_to_63,14);
S_Spare_1:=maskbitFunction(Trip_BITs_48_to_63,15);

T_Surge_detection:=maskbitFunction(Trip_BITs_64_to_79,0);
T_VGD_fault :=maskbitFunction(Trip_BITs_64_to_79,1);
T_Long_time_PRV :=maskbitFunction(Trip_BITs_64_to_79,2);
T_Comp_thrust_bearing_position :=maskbitFunction(Trip_BITs_64_to_79,3);
T_Comp_thrust_neg_move:=maskbitFunction(Trip_BITs_64_to_79,4);
T_Comp_thrust_pos_move:=maskbitFunction(Trip_BITs_64_to_79,5);
S_Spare_1:=maskbitFunction(Trip_BITs_64_to_79,6);
S_Spare_1:=maskbitFunction(Trip_BITs_64_to_79,7);
S_Spare_1:=maskbitFunction(Trip_BITs_64_to_79,8);
S_Spare_1:=maskbitFunction(Trip_BITs_64_to_79,9);
S_Spare_1:=maskbitFunction(Trip_BITs_64_to_79,10);
S_Spare_1:=maskbitFunction(Trip_BITs_64_to_79,11);
S_Spare_1:=maskbitFunction(Trip_BITs_64_to_79,12);
S_Spare_1:=maskbitFunction(Trip_BITs_64_to_79,13);
S_Spare_1:=maskbitFunction(Trip_BITs_64_to_79,14);
S_Spare_1:=maskbitFunction(Trip_BITs_64_to_79,15);

T_Sensor_low_signal_AI_64 :=maskbitFunction(Trip_BITs_80_to_95,0);
T_Sensor_high_signal_AI_64 :=maskbitFunction(Trip_BITs_80_to_95,1);
T_Sensor_low_signal_AI_66 :=maskbitFunction(Trip_BITs_80_to_95,2);
T_Sensor_high_signal_AI_66 :=maskbitFunction(Trip_BITs_80_to_95,3);
//T_Sensor_low_signal_AI_116:=maskbitFunction(Trip_BITs_80_to_95,4);
//T_Sensor_high_signal_AI_116:=maskbitFunction(Trip_BITs_80_to_95,5);
//T_Sensor_low_signal_AI_118:=maskbitFunction(Trip_BITs_80_to_95,6);
//T_Sensor_high_signal_AI_118:=maskbitFunction(Trip_BITs_80_to_95,7);
T_Sensor_low_signal_AI_128 :=maskbitFunction(Trip_BITs_80_to_95,8);
T_Sensor_high_signal_AI_128 :=maskbitFunction(Trip_BITs_80_to_95,9);
T_Sensor_low_signal_AI_130 :=maskbitFunction(Trip_BITs_80_to_95,10);
T_Sensor_high_signal_AI_130 :=maskbitFunction(Trip_BITs_80_to_95,11);
T_Sensor_low_signal_AI_132 :=maskbitFunction(Trip_BITs_80_to_95,12);
T_Sensor_high_signal_AI_132 :=maskbitFunction(Trip_BITs_80_to_95,13);
T_Sensor_low_signal_AI_134 :=maskbitFunction(Trip_BITs_80_to_95,14);
T_Sensor_high_signal_AI_134 :=maskbitFunction(Trip_BITs_80_to_95,15);

T_Sensor_low_signal_AI_136 :=maskbitFunction(Trip_BITs_96_to_121,0);
T_Sensor_high_signal_AI_136 :=maskbitFunction(Trip_BITs_96_to_121,1);
T_Sensor_low_signal_AI_138 :=maskbitFunction(Trip_BITs_96_to_121,2);
T_Sensor_high_signal_AI_138 :=maskbitFunction(Trip_BITs_96_to_121,3);
T_Sensor_low_signal_AI_140 :=maskbitFunction(Trip_BITs_96_to_121,4);
T_Sensor_high_signal_AI_140 :=maskbitFunction(Trip_BITs_96_to_121,5);
T_Sensor_low_signal_AI_142 :=maskbitFunction(Trip_BITs_96_to_121,6);
T_Sensor_high_signal_AI_142 :=maskbitFunction(Trip_BITs_96_to_121,7);
T_Sensor_low_signal_AI_144 :=maskbitFunction(Trip_BITs_96_to_121,8);
T_Sensor_high_signal_AI_144 :=maskbitFunction(Trip_BITs_96_to_121,9);
T_Sensor_low_signal_AI_146 :=maskbitFunction(Trip_BITs_96_to_121,10);
T_Sensor_high_signal_AI_146 :=maskbitFunction(Trip_BITs_96_to_121,11);
T_Sensor_low_signal_AI_148 :=maskbitFunction(Trip_BITs_96_to_121,12);
T_Sensor_high_signal_AI_148 :=maskbitFunction(Trip_BITs_96_to_121,13);
T_Sensor_low_signal_AI_150 :=maskbitFunction(Trip_BITs_96_to_121,14);
T_Sensor_high_signal_AI_150 :=maskbitFunction(Trip_BITs_96_to_121,15);

T_Sensor_low_signal_AI_152 :=maskbitFunction(Trip_BITs_122_to_137,0);
T_Sensor_high_signal_AI_152 :=maskbitFunction(Trip_BITs_122_to_137,1);
T_Sensor_low_signal_AI_154 :=maskbitFunction(Trip_BITs_122_to_137,2);
T_Sensor_high_signal_AI_154 :=maskbitFunction(Trip_BITs_122_to_137,3);
T_Sensor_low_signal_AI_156 :=maskbitFunction(Trip_BITs_122_to_137,4);
T_Sensor_high_signal_AI_156 :=maskbitFunction(Trip_BITs_122_to_137,5);
T_Sensor_low_signal_AI_158 :=maskbitFunction(Trip_BITs_122_to_137,6);
T_Sensor_high_signal_AI_158 :=maskbitFunction(Trip_BITs_122_to_137,7);
T_Sensor_low_signal_AI_160 :=maskbitFunction(Trip_BITs_122_to_137,8);
T_Sensor_high_signal_AI_160 :=maskbitFunction(Trip_BITs_122_to_137,9);
T_Sensor_low_signal_AI_162 :=maskbitFunction(Trip_BITs_122_to_137,10);
T_Sensor_high_signal_AI_162 :=maskbitFunction(Trip_BITs_122_to_137,11);
T_Sensor_low_signal_AI_164 :=maskbitFunction(Trip_BITs_122_to_137,12);
T_Sensor_high_signal_AI_164 :=maskbitFunction(Trip_BITs_122_to_137,13);
T_Sensor_low_signal_AI_166 :=maskbitFunction(Trip_BITs_122_to_137,14);
T_Sensor_high_signal_AI_166 :=maskbitFunction(Trip_BITs_122_to_137,15);

T_Sensor_low_signal_AI_168 :=maskbitFunction(Trip_BITs_138_to_153,0);
T_Sensor_high_signal_AI_168 :=maskbitFunction(Trip_BITs_138_to_153,1);
T_Sensor_low_signal_AI_170 :=maskbitFunction(Trip_BITs_138_to_153,2);
T_Sensor_high_signal_AI_170:=maskbitFunction(Trip_BITs_138_to_153,3);
T_Sensor_high_signal_AI_172:=maskbitFunction(Trip_BITs_138_to_153,4);
T_Sensor_high_signal_AI_172:=maskbitFunction(Trip_BITs_138_to_153,5);
T_Sensor_high_signal_AI_174:=maskbitFunction(Trip_BITs_138_to_153,6);
T_Sensor_high_signal_AI_174:=maskbitFunction(Trip_BITs_138_to_153,7);
T_Sensor_high_signal_AI_176:=maskbitFunction(Trip_BITs_138_to_153,8);
T_Sensor_high_signal_AI_176:=maskbitFunction(Trip_BITs_138_to_153,9);
T_Sensor_high_signal_AI_178:=maskbitFunction(Trip_BITs_138_to_153,10);
T_Sensor_high_signal_AI_178:=maskbitFunction(Trip_BITs_138_to_153,11);
T_Sensor_high_signal_AI_180:=maskbitFunction(Trip_BITs_138_to_153,12);
T_Sensor_high_signal_AI_180:=maskbitFunction(Trip_BITs_138_to_153,13);
T_Sensor_high_signal_AI_182:=maskbitFunction(Trip_BITs_138_to_153,14);
T_Sensor_high_signal_AI_182:=maskbitFunction(Trip_BITs_138_to_153,15);

T_Sensor_low_signal_AI_184 :=maskbitFunction(Trip_BITs_154_to_169,0);
T_Sensor_high_signal_AI_184 :=maskbitFunction(Trip_BITs_154_to_169,1);
T_Sensor_low_signal_AI_186 :=maskbitFunction(Trip_BITs_154_to_169,2);
T_Sensor_high_signal_AI_186 :=maskbitFunction(Trip_BITs_154_to_169,3);
T_Sensor_low_signal_AI_188 :=maskbitFunction(Trip_BITs_154_to_169,4);
T_Sensor_high_signal_AI_188 :=maskbitFunction(Trip_BITs_154_to_169,5);
T_Sensor_low_signal_AI_190 :=maskbitFunction(Trip_BITs_154_to_169,6);
T_Sensor_high_signal_AI_190 :=maskbitFunction(Trip_BITs_154_to_169,7);
T_Sensor_low_signal_AI_192 :=maskbitFunction(Trip_BITs_154_to_169,8);
T_Sensor_high_signal_AI_192 :=maskbitFunction(Trip_BITs_154_to_169,9);
T_Sensor_low_signal_AI_194 :=maskbitFunction(Trip_BITs_154_to_169,10);
T_Sensor_high_signal_AI_194 :=maskbitFunction(Trip_BITs_154_to_169,11);
T_Sensor_low_signal_AI_196 :=maskbitFunction(Trip_BITs_154_to_169,12);
T_Sensor_high_signal_AI_196 :=maskbitFunction(Trip_BITs_154_to_169,13);
T_Sensor_low_signal_AI_198 :=maskbitFunction(Trip_BITs_154_to_169,14);
T_Sensor_high_signal_AI_198 :=maskbitFunction(Trip_BITs_154_to_169,15);

T_Sensor_low_signal_AI_200 :=maskbitFunction(Trip_BITs_170_to_185,0);
T_Sensor_high_signal_AI_200 :=maskbitFunction(Trip_BITs_170_to_185,1);
T_Sensor_low_signal_AI_202 :=maskbitFunction(Trip_BITs_170_to_185,2);
T_Sensor_high_signal_AI_202 :=maskbitFunction(Trip_BITs_170_to_185,3);
T_Sensor_low_signal_AI_204 :=maskbitFunction(Trip_BITs_170_to_185,4);
T_Sensor_high_signal_AI_204 :=maskbitFunction(Trip_BITs_170_to_185,5);
T_Sensor_low_signal_AI_206 :=maskbitFunction(Trip_BITs_170_to_185,6);
T_Sensor_high_signal_AI_206 :=maskbitFunction(Trip_BITs_170_to_185,7);
S_Spare_1:=maskbitFunction(Trip_BITs_170_to_185,8);
S_Spare_1 :=maskbitFunction(Trip_BITs_170_to_185,9);
S_Spare_1 :=maskbitFunction(Trip_BITs_170_to_185,10);
S_Spare_1 :=maskbitFunction(Trip_BITs_170_to_185,11);
S_Spare_1 :=maskbitFunction(Trip_BITs_170_to_185,12);
S_Spare_1 :=maskbitFunction(Trip_BITs_170_to_185,13);
S_Spare_1 :=maskbitFunction(Trip_BITs_170_to_185,14);
S_Spare_1 :=maskbitFunction(Trip_BITs_170_to_185,15);

T_Transformer_winding_temp :=maskbitFunction(Trip_BITs_186_to_201,0);
T_trafo_opening_main_breaker :=maskbitFunction(Trip_BITs_186_to_201,1);
S_Spare_1 :=maskbitFunction(Trip_BITs_186_to_201,2);
S_Spare_1 :=maskbitFunction(Trip_BITs_186_to_201,3);
S_Spare_1 :=maskbitFunction(Trip_BITs_186_to_201,4);
S_Spare_1 :=maskbitFunction(Trip_BITs_186_to_201,5);
S_Spare_1 :=maskbitFunction(Trip_BITs_186_to_201,6);
S_Spare_1 :=maskbitFunction(Trip_BITs_186_to_201,7);
S_Spare_1 :=maskbitFunction(Trip_BITs_186_to_201,8);
S_Spare_1 :=maskbitFunction(Trip_BITs_186_to_201,9);
S_Spare_1 :=maskbitFunction(Trip_BITs_186_to_201,10);
S_Spare_1 :=maskbitFunction(Trip_BITs_186_to_201,11);
S_Spare_1 :=maskbitFunction(Trip_BITs_186_to_201,12);
S_Spare_1 :=maskbitFunction(Trip_BITs_186_to_201,13);
S_Spare_1 :=maskbitFunction(Trip_BITs_186_to_201,14);
S_Spare_1 :=maskbitFunction(Trip_BITs_186_to_201,15);


// Alarm bits
A_low_disch_press:=maskbitFunction(Alarm_BITs_0_to_15,0);
A_high_disch_press:=maskbitFunction(Alarm_BITs_0_to_15,1);
A_Low_suction_pressure:=maskbitFunction(Alarm_BITs_0_to_15,2);
A_High_suction_pressure:=maskbitFunction(Alarm_BITs_0_to_15,3);
A_Low_press_ratio:=maskbitFunction(Alarm_BITs_0_to_15,4);
A_High_discharge_temp :=maskbitFunction(Alarm_BITs_0_to_15,5);
A_Low_discharge_superheat:=maskbitFunction(Alarm_BITs_0_to_15,6);
A_High_discharge_superheat:=maskbitFunction(Alarm_BITs_0_to_15,7);
S_Spare_1:=maskbitFunction(Alarm_BITs_0_to_15,8);
S_Spare_1:=maskbitFunction(Alarm_BITs_0_to_15,9);
A_Low_temp_oil_inlet_comp:=maskbitFunction(Alarm_BITs_0_to_15,10);
A_High_temp_oil_inlet_comp:=maskbitFunction(Alarm_BITs_0_to_15,11);
A_Low_oil_temp_receiver:=maskbitFunction(Alarm_BITs_0_to_15,12);
A_High_oil_temp_receiver:=maskbitFunction(Alarm_BITs_0_to_15,13);
A_Low_oil_diff_pressure:=maskbitFunction(Alarm_BITs_0_to_15,14);
A_High_oil_diff_pressure:=maskbitFunction(Alarm_BITs_0_to_15,15);

A_High_oil_filter_diff_press:=maskbitFunction(Alarm_BITs_16_to_31,0);
S_Spare_1:=maskbitFunction(Alarm_BITs_16_to_31,1);
S_Spare_1:=maskbitFunction(Alarm_BITs_16_to_31,2);
A_Low_CW_outlet_temp:=maskbitFunction(Alarm_BITs_16_to_31,3);
A_High_CW_inlet_temp:=maskbitFunction(Alarm_BITs_16_to_31,4);
A_Low_CW_dP:=maskbitFunction(Alarm_BITs_16_to_31,5);
A_High_CW_dP:=maskbitFunction(Alarm_BITs_16_to_31,6);
S_Spare_1:=maskbitFunction(Alarm_BITs_16_to_31,7);
S_Spare_1:=maskbitFunction(Alarm_BITs_16_to_31,8);
A_Low_SW_inlet_temp:=maskbitFunction(Alarm_BITs_16_to_31,9);
A_High_SW_inlet_temp:=maskbitFunction(Alarm_BITs_16_to_31,10);
A_Low_SW_dP:=maskbitFunction(Alarm_BITs_16_to_31,11);
A_High_SW_dP:=maskbitFunction(Alarm_BITs_16_to_31,12);
A_Low_liquid_level:=maskbitFunction(Alarm_BITs_16_to_31,13);
A_Seawater_pump_not_running:=maskbitFunction(Alarm_BITs_16_to_31,14);
S_Spare_1:=maskbitFunction(Alarm_BITs_16_to_31,15);

S_Spare_1:=maskbitFunction(Alarm_BITs_32_to_47,0);
A_High_motor_wind_temp_R:=maskbitFunction(Alarm_BITs_32_to_47,1);
A_High_motor_wind_temp_S:=maskbitFunction(Alarm_BITs_32_to_47,2);
A_High_motor_wind_temp_T:=maskbitFunction(Alarm_BITs_32_to_47,3);
A_High_comp_mo_DE_bear_temp:=maskbitFunction(Alarm_BITs_32_to_47,4);
A_High_comp_mo_NDE_bear_temp:=maskbitFunction(Alarm_BITs_32_to_47,5);
A_High_motor_air_temp:=maskbitFunction(Alarm_BITs_32_to_47,6); 
A_High_comp_mo_DE_bear_vib:=maskbitFunction(Alarm_BITs_32_to_47,7);
A_High_comp_mo_NDE_bear_vib:=maskbitFunction(Alarm_BITs_32_to_47,8);
S_Spare_1:=maskbitFunction(Alarm_BITs_32_to_47,9);
S_Spare_1:=maskbitFunction(Alarm_BITs_32_to_47,10);
A_VGD_fault:=maskbitFunction(Alarm_BITs_32_to_47,11);
A_High_control_panel_temp:=maskbitFunction(Alarm_BITs_32_to_47,12);
A_Suction_press_limit:=maskbitFunction(Alarm_BITs_32_to_47,13);
A_Discharge_press_limit:=maskbitFunction(Alarm_BITs_32_to_47,14);
A_Discharge_superheat_limit:=maskbitFunction(Alarm_BITs_32_to_47,15);

A_Motor_current_limit:=maskbitFunction(Alarm_BITs_48_to_63,0);
S_Spare_1:=maskbitFunction(Alarm_BITs_48_to_63,1);
S_Spare_1:=maskbitFunction(Alarm_BITs_48_to_63,2);
S_Spare_1:=maskbitFunction(Alarm_BITs_48_to_63,3);
S_Spare_1:=maskbitFunction(Alarm_BITs_48_to_63,4);
S_Spare_1:=maskbitFunction(Alarm_BITs_48_to_63,5);
S_Spare_1:=maskbitFunction(Alarm_BITs_48_to_63,6);
S_Spare_1:=maskbitFunction(Alarm_BITs_48_to_63,7);
S_Spare_1:=maskbitFunction(Alarm_BITs_48_to_63,8);
S_Spare_1:=maskbitFunction(Alarm_BITs_48_to_63,9);
S_Spare_1:=maskbitFunction(Alarm_BITs_48_to_63,10);
S_Spare_1:=maskbitFunction(Alarm_BITs_48_to_63,11);
S_Spare_1:=maskbitFunction(Alarm_BITs_48_to_63,12);
S_Spare_1:=maskbitFunction(Alarm_BITs_48_to_63,13);
S_Spare_1:=maskbitFunction(Alarm_BITs_48_to_63,14);
S_Spare_1:=maskbitFunction(Alarm_BITs_48_to_63,15);

A_Transformer_winding_temp:=maskbitFunction(Alarm_BITs_64_to_79,0);
S_Spare_1:=maskbitFunction(Alarm_BITs_64_to_79,1);
S_Spare_1:=maskbitFunction(Alarm_BITs_64_to_79,2);
S_Spare_1:=maskbitFunction(Alarm_BITs_64_to_79,3);
S_Spare_1:=maskbitFunction(Alarm_BITs_64_to_79,4);
S_Spare_1:=maskbitFunction(Alarm_BITs_64_to_79,5);
S_Spare_1:=maskbitFunction(Alarm_BITs_64_to_79,6);
S_Spare_1:=maskbitFunction(Alarm_BITs_64_to_79,7);
S_Spare_1:=maskbitFunction(Alarm_BITs_64_to_79,8);
S_Spare_1:=maskbitFunction(Alarm_BITs_64_to_79,9);
S_Spare_1:=maskbitFunction(Alarm_BITs_64_to_79,10);
S_Spare_1:=maskbitFunction(Alarm_BITs_64_to_79,11);
S_Spare_1:=maskbitFunction(Alarm_BITs_64_to_79,12);
S_Spare_1:=maskbitFunction(Alarm_BITs_64_to_79,13);
S_Spare_1:=maskbitFunction(Alarm_BITs_64_to_79,14);
S_Spare_1:=maskbitFunction(Alarm_BITs_64_to_79,15);

// Statusbits
DI_0_0_Emergency_stop:=maskbitFunction(Status_BITs_0_to_15,0);
Unit_start_switch:=maskbitFunction(Status_BITs_0_to_15,1);
DI_0_2_Fault_reset:=maskbitFunction(Status_BITs_0_to_15,2);
Unit_auto:=maskbitFunction(Status_BITs_0_to_15,3);
Unit_remote:=maskbitFunction(Status_BITs_0_to_15,4);
Unit_manual:=maskbitFunction(Status_BITs_0_to_15,5);
DI_0_6_Overload_protection:=maskbitFunction(Status_BITs_0_to_15,6);
Unit_running:=maskbitFunction(Status_BITs_0_to_15,7);
DI_1_0_Overload_oilpump:=maskbitFunction(Status_BITs_0_to_15,8);
Comp_oil_pump:=maskbitFunction(Status_BITs_0_to_15,9);
Sea_water_pump:=maskbitFunction(Status_BITs_0_to_15,10);
CW_pump_running:=maskbitFunction(Status_BITs_0_to_15,11);
DI_1_4_Power_available:=maskbitFunction(Status_BITs_0_to_15,12);
DI_1_5_Starter_failure:=maskbitFunction(Status_BITs_0_to_15,13);
//CW_Pump_Remote_Start_Available:=maskbitFunction(Status_BITs_0_to_15,14);
//T_CW_Pump:=maskbitFunction(Status_BITs_0_to_15,15);

DI_8_0_Controlpanel_temp:=maskbitFunction(Status_BITs_16_to_31,0);
CW_Flow_ind:=maskbitFunction(Status_BITs_16_to_31,1);
DI_8_2_VGD_limit_switch:=maskbitFunction(Status_BITs_16_to_31,2);
DI_8_3_water_leak_motor:=maskbitFunction(Status_BITs_16_to_31,3);
DI_8_4_Catodic_protection:=maskbitFunction(Status_BITs_16_to_31,4);
DI_8_5_Trust_bearing_probe:=maskbitFunction(Status_BITs_16_to_31,5);
DI_8_6_ESD_operation:=maskbitFunction(Status_BITs_16_to_31,6);
DI_8_7:=maskbitFunction(Status_BITs_16_to_31,7);
DI_9_0_MV_breaker_available:=maskbitFunction(Status_BITs_16_to_31,8);
DI_9_1:=maskbitFunction(Status_BITs_16_to_31,9);
DI_9_2_Safe_return_to_port:=maskbitFunction(Status_BITs_16_to_31,10);
VFD_ready:=maskbitFunction(Status_BITs_16_to_31,11);
DI_9_4_VFD_emergency_stop:=maskbitFunction(Status_BITs_16_to_31,12);
Remote_bilge_pump_control:=maskbitFunction(Status_BITs_16_to_31,13);
//T_Transformer:=maskbitFunction(Status_BITs_16_to_31,14);
//A_Transformer:=maskbitFunction(Status_BITs_16_to_31,15);

DO_0_0_Start_signal_comp:=maskbitFunction(Status_BITs_32_to_47,0);
DO_0_1_Start_signal_oil_pump:=maskbitFunction(Status_BITs_32_to_47,1);
DO_0_2_Start_signal_SW_pump:=maskbitFunction(Status_BITs_32_to_47,2);
DO_0_3_Start_signal_CW_pump:=maskbitFunction(Status_BITs_32_to_47,3);
DO_0_4_Solenoid_valve_oil:=maskbitFunction(Status_BITs_32_to_47,4);
DO_0_5_Solenoid_valve_liquid:=maskbitFunction(Status_BITs_32_to_47,5);
DO_0_6_Oil_heater:=maskbitFunction(Status_BITs_32_to_47,6);
DO_0_7_Comp_heater:=maskbitFunction(Status_BITs_32_to_47,7);
DO_1_0:=maskbitFunction(Status_BITs_32_to_47,8);
DO_1_1:=maskbitFunction(Status_BITs_32_to_47,9);
S_Spare_1:=maskbitFunction(Status_BITs_32_to_47,10);
S_Spare_1:=maskbitFunction(Status_BITs_32_to_47,11);
S_Spare_1:=maskbitFunction(Status_BITs_32_to_47,12);
S_Spare_1:=maskbitFunction(Status_BITs_32_to_47,13);
S_Spare_1:=maskbitFunction(Status_BITs_32_to_47,14);
S_Spare_1:=maskbitFunction(Status_BITs_32_to_47,15);

DO_8_0_Liquid_valve_open:=maskbitFunction(Status_BITs_48_to_63,0);
DO_8_1_Liquid_valve_close:=maskbitFunction(Status_BITs_48_to_63,1);
DO_8_2_VGD_open:=maskbitFunction(Status_BITs_48_to_63,2);
DO_8_3_VGD_close:=maskbitFunction(Status_BITs_48_to_63,3);
DO_8_4_PRV_open:=maskbitFunction(Status_BITs_48_to_63,4);
DO_8_5_PRV_close:=maskbitFunction(Status_BITs_48_to_63,5);
DO_8_6_HGV_open:=maskbitFunction(Status_BITs_48_to_63,6);
DO_8_7_HGV_close:=maskbitFunction(Status_BITs_48_to_63,7);
DO_9_0_Main_breaker_ready:=maskbitFunction(Status_BITs_48_to_63,8);
DO_9_1_Close_order_swv_overboard:=maskbitFunction(Status_BITs_48_to_63,9);
DO_9_2_Open_order_swv_bypass:=maskbitFunction(Status_BITs_48_to_63,10);
DO_9_3_Close_order_swv_bypass:=maskbitFunction(Status_BITs_48_to_63,11);
DO_9_4:=maskbitFunction(Status_BITs_48_to_63,12);
DO_9_5:=maskbitFunction(Status_BITs_48_to_63,13);
DO_9_6:=maskbitFunction(Status_BITs_48_to_63,14);
DO_9_7:=maskbitFunction(Status_BITs_48_to_63,15);

DO_12_0_Power_request:=maskbitFunction(Status_BITs_64_to_79,0);
DO_12_1_Compressor_ready:=maskbitFunction(Status_BITs_64_to_79,1);
Unit_trip:=maskbitFunction(Status_BITs_64_to_79,2);
Unit_alarm:=maskbitFunction(Status_BITs_64_to_79,3);
DO_12_4_Control_panel_alarm:=maskbitFunction(Status_BITs_64_to_79,4);
DO_12_5_Auto_reset:=maskbitFunction(Status_BITs_64_to_79,5);
DO_12_6_Unit_running:=maskbitFunction(Status_BITs_64_to_79,6);
//DO_12_7_Emergency_MV_Breaker:=maskbitFunction(Status_BITs_64_to_79,7);
T_Spare_3:=maskbitFunction(Status_BITs_64_to_79,8);
T_Spare_3:=maskbitFunction(Status_BITs_64_to_79,9);
T_Spare_3:=maskbitFunction(Status_BITs_64_to_79,10);
T_Spare_3:=maskbitFunction(Status_BITs_64_to_79,11);
T_Spare_3:=maskbitFunction(Status_BITs_64_to_79,12);
T_Spare_3:=maskbitFunction(Status_BITs_64_to_79,13);
T_Spare_3:=maskbitFunction(Status_BITs_64_to_79,14);
T_Spare_3:=maskbitFunction(Status_BITs_64_to_79,15);

Unit_manual:=maskbitFunction(Status_BITs_80_to_95,0);
Unit_available:=maskbitFunction(Status_BITs_80_to_95,1);
CW_Flow_ind:=maskbitFunction(Status_BITs_80_to_95,2);
Start_inhib_time_Oil_receiver_temp:=maskbitFunction(Status_BITs_80_to_95,3);
Start_inhib_time_between_Stop_Start:=maskbitFunction(Status_BITs_80_to_95,4);
Start_inhib_time_between_Start:=maskbitFunction(Status_BITs_80_to_95,5);
Start_inhib_PRV_not_min:=maskbitFunction(Status_BITs_80_to_95,6);
VFD_ramp_100_perc:=maskbitFunction(Status_BITs_80_to_95,7);
VFD_locked_100_perc:=maskbitFunction(Status_BITs_80_to_95,8);
VFD_ramp_d_PRVcontrol:=maskbitFunction(Status_BITs_80_to_95,9);
PRV_control:=maskbitFunction(Status_BITs_80_to_95,10);
VFD_control:=maskbitFunction(Status_BITs_80_to_95,11);
VFD_fixed_speed:=maskbitFunction(Status_BITs_80_to_95,12);
T_Spare_3:=maskbitFunction(Status_BITs_80_to_95,13);
T_Spare_3:=maskbitFunction(Status_BITs_80_to_95,14);
T_Spare_3:=maskbitFunction(Status_BITs_80_to_95,15);


// Graphic controls
IF Unit_remote THEN
	Unit_switch_status:=2;
ELSIF Unit_auto THEN 
	Unit_switch_status:=3;
ELSIF Unit_manual THEN 
	Unit_switch_status:=4;

END_IF ;	

IF select_trendvalue > 0 THEN
	show_trendvalue[select_trendvalue]:= TRUE;
ELSIF select_trendvalue = 0 THEN
	FOR i := 0 TO 50 DO
      show_trendvalue[i] := FALSE;
   	END_FOR
END_IF ;

END_PROGRAM

// Chiller_2
PROGRAM Chiller_2
VAR

timer2 : standard.ton ;
{attribute 'ac_datalog_set_default_group' := 'DataLogChannel_2'}
instStruct : LogStruct;


modbus_var : ARRAY[0..100] OF INT;
modbus_var_1000 : ARRAY[0..123] OF WORD;
modbus_var_1001 : ARRAY[124..247] OF WORD;
modbus_var_1002 : ARRAY[248..371] OF WORD;
{attribute 'ac_datalog_hysteresis' := '0.2'}
{attribute 'ac_datalog' := 'DataLogChannel_2'}
Temp_chilled_medium_out : REAL;
{attribute 'ac_datalog_hysteresis' := '0.2'}
{attribute 'ac_datalog' := 'DataLogChannel_2'}
Temp_chilled_medium_in : REAL;
{attribute 'ac_datalog_hysteresis' := '0.2'}
{attribute 'ac_datalog' := 'DataLogChannel_2'}
Temp_water_inlet_cond : REAL;
{attribute 'ac_datalog_hysteresis' := '0.2'}
{attribute 'ac_datalog' := 'DataLogChannel_2'}
Press_suction_compr : REAL;
{attribute 'ac_datalog_hysteresis' := '0.5'}
{attribute 'ac_datalog' := 'DataLogChannel_2'}
Press_discharge_compr : REAL;
{attribute 'ac_datalog_hysteresis' := '0.5'}
{attribute 'ac_datalog' := 'DataLogChannel_2'}
Press_oil_receiver : REAL;
{attribute 'ac_datalog_hysteresis' := '0.5'}
{attribute 'ac_datalog' := 'DataLogChannel_2'}
Press_oil_compr : REAL;
{attribute 'ac_datalog_hysteresis' := '0.4'}
{attribute 'ac_datalog' := 'DataLogChannel_2'}
Temp_discharge : REAL;
{attribute 'ac_datalog_hysteresis' := '0.5'}
{attribute 'ac_datalog' := 'DataLogChannel_2'}
Oil_temp_receiver : REAL;
{attribute 'ac_datalog_hysteresis' := '0.5'}
{attribute 'ac_datalog' := 'DataLogChannel_2'}
Max_motor_temp : REAL;
{attribute 'ac_datalog_hysteresis' := '0.2'}
{attribute 'ac_datalog' := 'DataLogChannel_2'}
Temp_motor_bearing_DE : REAL;
{attribute 'ac_datalog_hysteresis' := '0.2'}
{attribute 'ac_datalog' := 'DataLogChannel_2'}
Temp_motor_bearing_NDE : REAL;
{attribute 'ac_datalog_hysteresis' := '4'}
{attribute 'ac_datalog' := 'DataLogChannel_2'}
Motor_current : REAL;
{attribute 'ac_datalog_hysteresis' := '50'}
{attribute 'ac_datalog' := 'DataLogChannel_2'}
Running_hours_comp_unscaled : WORD;
{attribute 'ac_datalog_hysteresis' := '50'}
{attribute 'ac_datalog' := 'DataLogChannel_2'}
Running_hours_oil_pump_unscaled : WORD;
{attribute 'ac_datalog' := 'DataLogChannel_2'}
Anti_recycle_time : REAL;
{attribute 'ac_datalog_hysteresis' := '2'}
{attribute 'ac_datalog' := 'DataLogChannel_2'}
Feedback_compressor : REAL;
{attribute 'ac_datalog_hysteresis' := '0.2'}
{attribute 'ac_datalog' := 'DataLogChannel_2'}
Oil_diff_pressure : REAL;
{attribute 'ac_datalog_hysteresis' := '0.3'}
{attribute 'ac_datalog' := 'DataLogChannel_2'}
Suction_saturated_temp : REAL;
{attribute 'ac_datalog_hysteresis' := '0.2'}
{attribute 'ac_datalog' := 'DataLogChannel_2'}
Discharge_saturated_temp : REAL;
{attribute 'ac_datalog_hysteresis' := '0.2'}
{attribute 'ac_datalog' := 'DataLogChannel_2'}
Temp_water_outlet_cond : REAL;
{attribute 'ac_datalog_hysteresis' := '0.2'}
{attribute 'ac_datalog' := 'DataLogChannel_2'}
Temp_motor_wind_R : REAL;
{attribute 'ac_datalog_hysteresis' := '0.2'}
{attribute 'ac_datalog' := 'DataLogChannel_2'}
Temp_motor_wind_S : REAL;
{attribute 'ac_datalog_hysteresis' := '0.2'}
{attribute 'ac_datalog' := 'DataLogChannel_2'}
Temp_motor_wind_T : REAL;
{attribute 'ac_datalog_hysteresis' := '0.2'}
{attribute 'ac_datalog' := 'DataLogChannel_2'}
Temp_motor_air : REAL;
{attribute 'ac_datalog_hysteresis' := '0.04'}
{attribute 'ac_datalog' := 'DataLogChannel_2'}
dP_CW : REAL;
{attribute 'ac_datalog_hysteresis' := '0.04'}
{attribute 'ac_datalog' := 'DataLogChannel_2'}
dP_SW : REAL;
{attribute 'ac_datalog_hysteresis' := '4'}
{attribute 'ac_datalog' := 'DataLogChannel_2'}
Chiller_capacity : REAL;
{attribute 'ac_datalog_hysteresis' := '2'}
{attribute 'ac_datalog' := 'DataLogChannel_2'}
Temp_oil_inlet_compr : REAL;
Spare : REAL;
{attribute 'ac_datalog_hysteresis' := '2'}
{attribute 'ac_datalog' := 'DataLogChannel_2'}
SP_CW_controller : REAL;
{attribute 'ac_datalog_hysteresis' := '2'}
{attribute 'ac_datalog' := 'DataLogChannel_2'}
Setpoint_oil_pump : REAL;
{attribute 'ac_datalog_hysteresis' := '0.02'}
{attribute 'ac_datalog' := 'DataLogChannel_2'}
Thrust_bearing_position : REAL;
{attribute 'ac_datalog_hysteresis' := '50'}
{attribute 'ac_datalog' := 'DataLogChannel_2'}
Oil_pump_running_hours : REAL;
{attribute 'ac_datalog_hysteresis' := '5'}
{attribute 'ac_datalog' := 'DataLogChannel_2'}
Liquid_level_condenser : REAL;
{attribute 'ac_datalog_hysteresis' := '0.05'}
{attribute 'ac_datalog' := 'DataLogChannel_2'}
Oil_Filter_Drop : REAL; 
{attribute 'ac_datalog_hysteresis' := '2'}
{attribute 'ac_datalog' := 'DataLogChannel_2'}
Proximitor_thrust_pos : REAL;
{attribute 'ac_datalog_hysteresis' := '0.4'}
{attribute 'ac_datalog' := 'DataLogChannel_2'}
Press_chilled_medium_in : REAL;
{attribute 'ac_datalog_hysteresis' := '0.2'}
{attribute 'ac_datalog' := 'DataLogChannel_2'}
Press_water_cond_out : REAL;
{attribute 'ac_datalog_hysteresis' := '0.02'}
{attribute 'ac_datalog' := 'DataLogChannel_2'}
Feedback_sea_water_valve : REAL;
{attribute 'ac_datalog_hysteresis' := '1'}
{attribute 'ac_datalog' := 'DataLogChannel_2'}
Oil_pressure_before_filter : REAL;
{attribute 'ac_datalog_hysteresis' := '0.2'}
{attribute 'ac_datalog' := 'DataLogChannel_2'}
Trafo_winding_temp : REAL;
{attribute 'ac_datalog_hysteresis' := '1'}
{attribute 'ac_datalog' := 'DataLogChannel_2'}
Feedback_VGD : REAL;
{attribute 'ac_datalog_hysteresis' := '4'}
{attribute 'ac_datalog' := 'DataLogChannel_2'}
Feedback_liquid_valve : REAL;
{attribute 'ac_datalog_hysteresis' := '3'}
{attribute 'ac_datalog' := 'DataLogChannel_2'}
Feedback_HGV : REAL;
{attribute 'ac_datalog_hysteresis' := '2'}
{attribute 'ac_datalog' := 'DataLogChannel_2'}
Discharge_superheat : REAL;
{attribute 'ac_datalog_hysteresis' := '0.6'}
{attribute 'ac_datalog' := 'DataLogChannel_2'}
Frequency_oil_pump : REAL;
{attribute 'ac_datalog_hysteresis' := '3'}
{attribute 'ac_datalog' := 'DataLogChannel_2'}
Hot_gas_valve_output : REAL;
{attribute 'ac_datalog_hysteresis' := '2'}
{attribute 'ac_datalog' := 'DataLogChannel_2'}
Control_signal_unit_d : REAL;
{attribute 'ac_datalog_hysteresis' := '2'}
{attribute 'ac_datalog' := 'DataLogChannel_2'}
Stall_detector : REAL;
{attribute 'ac_datalog_hysteresis' := '0.2'}
{attribute 'ac_datalog' := 'DataLogChannel_2'}
SP_MC_controller : REAL;
{attribute 'ac_datalog_hysteresis' := '2'}
{attribute 'ac_datalog' := 'DataLogChannel_2'}
Prerotary_output : REAL;
{attribute 'ac_datalog_hysteresis' := '2'}
{attribute 'ac_datalog' := 'DataLogChannel_2'}
VGD_output : REAL;
{attribute 'ac_datalog_hysteresis' := '2'}
{attribute 'ac_datalog' := 'DataLogChannel_2'}
SP_PID_compressor : REAL;
{attribute 'ac_datalog_hysteresis' := '2'}
{attribute 'ac_datalog' := 'DataLogChannel_2'}
Output_PID_suction : REAL;
{attribute 'ac_datalog_hysteresis' := '2'}
{attribute 'ac_datalog' := 'DataLogChannel_2'}
Output_PID_discharge : REAL;
{attribute 'ac_datalog_hysteresis' := '2'}
{attribute 'ac_datalog' := 'DataLogChannel_2'}
Output_PID_motor : REAL;
{attribute 'ac_datalog_hysteresis' := '2'}
{attribute 'ac_datalog' := 'DataLogChannel_2'}
Output_PID_superheat : REAL;
{attribute 'ac_datalog_hysteresis' := '2'}
{attribute 'ac_datalog' := 'DataLogChannel_2'}
SP_control : REAL;
{attribute 'ac_datalog_hysteresis' := '2'}
{attribute 'ac_datalog' := 'DataLogChannel_2'}
Unit_control_signal : REAL;
{attribute 'ac_datalog_hysteresis' := '2'}
{attribute 'ac_datalog' := 'DataLogChannel_2'}
Feedback_PRV : REAL;
{attribute 'ac_datalog_hysteresis' := '0.3'}
{attribute 'ac_datalog' := 'DataLogChannel_2'}
Theta_out : REAL;
{attribute 'ac_datalog_hysteresis' := '50'}
{attribute 'ac_datalog' := 'DataLogChannel_2'}
Alarm_limit_stall_count_unscaled : WORD;
{attribute 'ac_datalog_hysteresis' := '50'}
{attribute 'ac_datalog' := 'DataLogChannel_2'}
Alarm_limit_stall_count : REAL;
{attribute 'ac_datalog_hysteresis' := '2'}
{attribute 'ac_datalog' := 'DataLogChannel_2'}
Stall_ramp : REAL;
Min_allowed_PRVposition : REAL;
Number_of_starts : REAL;
SP_oil_pressure : REAL;
{attribute 'ac_datalog_hysteresis' := '2'}
{attribute 'ac_datalog' := 'DataLogChannel_2'}
Setpoint_conv_oil_pump : REAL;
Days_above_stall_limit : REAL;
Hrs_above_stall_limit : REAL;
Min_above_stall_limit : REAL;
Sec_above_stall_limit : REAL;
{attribute 'ac_datalog_hysteresis' := '2'}
{attribute 'ac_datalog' := 'DataLogChannel_2'}
SP_cond_press : REAL;
{attribute 'ac_datalog_hysteresis' := '2'}
{attribute 'ac_datalog' := 'DataLogChannel_2'}
SP_PID_Level : REAL;
{attribute 'ac_datalog_hysteresis' := '2'}
{attribute 'ac_datalog' := 'DataLogChannel_2'}
Control_signal_SW_valve : REAL;
{attribute 'ac_datalog_hysteresis' := '4'}
{attribute 'ac_datalog' := 'DataLogChannel_2'}
Liquid_valve_output : REAL;
{attribute 'ac_datalog_hysteresis' := '0.2'}
{attribute 'ac_datalog' := 'DataLogChannel_2'}
SP_PID_seawater : REAL;
{attribute 'ac_datalog_hysteresis' := '4'}
{attribute 'ac_datalog' := 'DataLogChannel_2'}
Chiller_capacity_t1 : REAL;
{attribute 'ac_datalog_hysteresis' := '2'}
{attribute 'ac_datalog' := 'DataLogChannel_2'}
SW_pump_speed_order : REAL;
{attribute 'ac_datalog_hysteresis' := '0.4'}
{attribute 'ac_datalog' := 'DataLogChannel_2'}
Press_chilled_medium_out : REAL;
{attribute 'ac_datalog_hysteresis' := '50'}
{attribute 'ac_datalog' := 'DataLogChannel_2'}
Running_hours_compressormotor : REAL;
{attribute 'ac_datalog_hysteresis' := '0.2'}
{attribute 'ac_datalog' := 'DataLogChannel_2'}
Press_water_cond_inlet : REAL;
{attribute 'ac_datalog_hysteresis' := '20'}
{attribute 'ac_datalog' := 'DataLogChannel_2'}
Speed_feedback_VFD : REAL;
{attribute 'ac_datalog_hysteresis' := '20'}
{attribute 'ac_datalog' := 'DataLogChannel_2'}
Order_VFD_perc : REAL;
{attribute 'ac_datalog_hysteresis' := '20'}
{attribute 'ac_datalog' := 'DataLogChannel_2'}
Order_VFD_Hz : REAL;
{attribute 'ac_datalog_hysteresis' := '20'}
{attribute 'ac_datalog' := 'DataLogChannel_2'}
Temp_trafo_wind_U : REAL;
{attribute 'ac_datalog_hysteresis' := '0.2'}
{attribute 'ac_datalog' := 'DataLogChannel_2'}
Temp_trafo_wind_V : REAL;
{attribute 'ac_datalog_hysteresis' := '0.2'}
{attribute 'ac_datalog' := 'DataLogChannel_2'}
Temp_trafo_wind_W : REAL;
{attribute 'ac_datalog_hysteresis' := '2'}
{attribute 'ac_datalog' := 'DataLogChannel_2'}
Opt_speed_VFD_perc : REAL;
{attribute 'ac_datalog_hysteresis' := '20'}
{attribute 'ac_datalog' := 'DataLogChannel_2'}
Opt_speed_VFD_Hz : REAL;
Surge_counter_VFD : REAL;
Spare_4 : REAL;
Spare_3 : REAL;
Spare_2 : REAL;
Spare_0 : REAL;
Vibration_compressor_DE: REAL;
Vibration_compressor_NDE: REAL;
Feedback_seawater_valve_overboard : REAL;
Feedback_seawater_valve_bypass : REAL;
CW_flow_m3: REAL;
SW_flow_m3: REAL;
Max_motor_wind_temp: REAL;
Order_SWW_overboard: REAL;
Order_SWW_bypass: REAL;
{attribute 'ac_datalog_hysteresis' := '0.4'}
{attribute 'ac_datalog' := 'DataLogChannel'}
COP_chiller_mech : REAL ;
{attribute 'ac_datalog_hysteresis' := '10'}
{attribute 'ac_datalog' := 'DataLogChannel'}
P2_mot_1_kW : REAL ;
{attribute 'ac_datalog_hysteresis' := '20'}
{attribute 'ac_datalog' := 'DataLogChannel'}
P1_motor_kW : REAL ;
{attribute 'ac_datalog_hysteresis' := '0.4'}
{attribute 'ac_datalog' := 'DataLogChannel'}
COP_chiller_ele : REAL ;
{attribute 'ac_datalog_hysteresis' := '0.2'}
{attribute 'ac_datalog' := 'DataLogChannel'}
PI_chiller : REAL ;
{attribute 'ac_datalog_hysteresis' := '40'}
{attribute 'ac_datalog' := 'DataLogChannel'}
Wasted_energy_kW : REAL ;
{attribute 'ac_datalog_hysteresis' := '200'}
{attribute 'ac_datalog' := 'DataLogChannel'}
Chiller_capacity_kW : REAL;
Thrust_bearing_ref_min : REAL ;
Thrust_bearing_ref_max : REAL ;
Thrust_bearing_ref : REAL ;
Q2_chillerMWh : REAL ;
Chiller_P1_MWh : REAL ;
Cal_date_MMYY : REAL ;
Chiller_P2_MWh : REAL ;
Liquid_line_temp : REAL ;
VFD_motor_current : REAL ;
Feedback_liquid_valve_raw : REAL ;
Feedback_VGD_raw : REAL ;
Feedback_PRV_raw : REAL ;
Feedback_HGV_raw : REAL ;
Feedback_seawater_valve_overboard_raw : REAL ;
Feedback_seawater_valve_bypass_raw : REAL ;
SP_cond_press_limit : REAL ;
SP_evap_press_limit : REAL ;
SP_discharge_superheat_limit : REAL ;
VFD_min_allowed_frequence : REAL ;
VFD_min_allowed_speed : REAL ;
CW_Pump_Speed_SP : REAL;

Trip_BITs_0_to_15 : WORD;
Trip_BITs_16_to_31: WORD;
Trip_BITs_32_to_47: WORD;
Trip_BITs_48_to_63: WORD;
Trip_BITs_64_to_79: WORD;
Trip_BITs_80_to_95: WORD;
Trip_BITs_96_to_121: WORD;
Trip_BITs_122_to_137: WORD;
Trip_BITs_138_to_153: WORD;
Trip_BITs_154_to_169: WORD;
Trip_BITs_170_to_185: WORD;
Trip_BITs_186_to_201: WORD;


Alarm_BITs_0_to_15: WORD;
Alarm_BITs_16_to_31: WORD;
Alarm_BITs_32_to_47: WORD;
Alarm_BITs_48_to_63: WORD;
Alarm_BITs_64_to_79: WORD;
Status_BITs_0_to_15 : WORD;
Status_BITs_16_to_31 : WORD;
Status_BITs_32_to_47: WORD;
Status_BITs_48_to_63: WORD;
Status_BITs_64_to_79: WORD;
Status_BITs_80_to_95: WORD;




DIStatusbits_0_to_15 : WORD;
DIStatusbits_16_to_31: WORD;

DOStatusbits_16_to_31: WORD;
DOStatusbits_32_to_47: WORD;

T_Overload_compressor_motor : BOOL;
T_Compressor_running_failure : BOOL;

T_Low_oil_flow : BOOL;
T_Overload_oil_pump_motor : BOOL;
T_Oil_pump_running_failure : BOOL;
T_Low_oil_flow_trip : BOOL;
T_High_temp_oil_receiver : BOOL;
T_Low_temp_oil_receiver : BOOL;
T_Low_suction_pressure : BOOL;
T_High_suction_pressure : BOOL;
T_High_discharge_pressure : BOOL;
T_Low_discharge_pressure : BOOL;
T_High_discharge_temp : BOOL;
T_Low_oil_diff_pressure : BOOL;
T_High_diff_oil_pressure : BOOL;
T_Starting_to_long : BOOL;
T_Surge_detection : BOOL;
T_Comp_thrust_bearing_position : BOOL;
Spare_trip_1 : BOOL;
T_Chilled_pump_run_failure : BOOL;
T_Sea_water_pump_run_failure : BOOL;
T_Low_chilled_medium_flow : BOOL;
T_High_chilled_medium_flow : BOOL;
T_Low_condenser_flow : BOOL;
T_High_condenser_flow : BOOL;
T_Emergency_stop : BOOL;
T_High_comp_mot_DE_bear_temp : BOOL;
T_High_comp_mot_NDE_bear_temp : BOOL;
T_High_motor_air_temp : BOOL;
T_Comp_motor_leak_detection : BOOL;
T_High_comp_mot_DE_bear_vib : BOOL;
T_High_comp_mot_NDE_bear_Vib : BOOL;
Spare_trip_2 : BOOL;
T_Rotating_stall_trip : BOOL;
T_Analog_inputs : BOOL;
T_Feedback_CW_valve : BOOL;
T_Low_oil_diff_press_prelub : BOOL;
T_Low_oil_diff_press_standstil : BOOL;

T_Spare_3 : BOOL;
T_Spare_4 : BOOL;
T_Spare_5 : BOOL;
T_Spare_6 : BOOL;
T_Spare_7 : BOOL;
T_Spare_8 : BOOL;
T_High_temp_oil_inlet_comp : BOOL;
T_Comp_motor_power_loss : BOOL;
Spare_trip_3 : BOOL;
T_Cathodic_protect_sys_alarm : BOOL;
T_High_oil_filter_diff_press : BOOL;
T_Flow_switch_FT01 : BOOL;
T_Starter_failure_trip : BOOL;
T_Incorrect_feedback_starter_trip : BOOL;


A_High_condenser_flow : BOOL;
A_Rotating_stall : BOOL;
A_High_temp_oil_inlet_comp : BOOL;
SpareAlarm_1 : BOOL;
A_High_motor_air_temp : BOOL;
A_High_control_panel_temp : BOOL;
A_Low_oil_diff_pressure : BOOL;
Spare_alarm_2 : BOOL;
A_High_comp_motor_winding_temp : BOOL;
A_High_comp_mo_DE_bear_temp : BOOL;
A_High_comp_mo_NDE_bear_temp : BOOL;
A_High_comp_mo_DE_bear_vib : BOOL;
A_High_comp_mo_NDE_bear_vib : BOOL;
A_Low_chilled_medium_flow : BOOL;
A_High_chilled_medium_flow : BOOL;
A_Low_sea_water_flow : BOOL;
A_Seawater_pump_not_running : BOOL;
A_Spare : BOOL;
A_Spare_1 : BOOL;
A_Spare_2 : BOOL;
A_Spare_3 : BOOL;
A_Spare_4 : BOOL;
A_Spare_5 : BOOL;
A_Spare_6 : BOOL;
A_Spare_7 : BOOL;
A_Spare_8 : BOOL;
A_Spare_9 : BOOL;
A_Spare_10 : BOOL;
A_Spare_11 : BOOL;
A_High_oil_filter_diff_press : BOOL;
A_Spare_12 : BOOL;
A_Spare_13 : BOOL;
A_Spare_14 : BOOL;
A_Spare_15 : BOOL;
A_Spare_16 : BOOL;
A_Spare_17 : BOOL;
Anti_recycle_status : BOOL;
Low_oil_temperature : BOOL;
Low_oil_temp_auto : BOOL;
Oil_heater : BOOL;
Sea_water_pump : BOOL;
Comp_oil_pump : BOOL;
Bearing_oil_pump : BOOL;
Solenoid_oil_return : BOOL;
Unit_running : BOOL;
Unit_remote : BOOL;
Unit_auto : BOOL;
Unit_manual : BOOL;
Unit_trip : BOOL;
Unit_alarm : BOOL;
Unit_start_switch : BOOL;
Unit_available : BOOL;
S_Spare_1 : BOOL;
S_Spare_2 : BOOL;
S_Spare_3 : BOOL;
S_Spare_4 : BOOL;
S_Spare_5 : BOOL;
S_Spare_6 : BOOL;
S_Spare_7 : BOOL;
S_Spare_8 : BOOL;
Solenoid_liquid_inj: BOOL;
CW_Flow_ind : BOOL;
Open_chilled_water_valve : BOOL;
Feedback_chilled_water_valve : BOOL;
Open_order_swv_overboard : BOOL;
Close_order_swv_overboard : BOOL;
Open_order_swv_bypass : BOOL;
Close_order_swv_bypass : BOOL;
VFD_man_auto : BOOL ;
VFD_freq_jump_on : BOOL ;
VFD_ramp_100_perc : BOOL ;
VFD_locked_100_perc : BOOL;
VFD_ramp_d_PRVcontrol : BOOL;
PRV_control : BOOL;
VFD_control : BOOL;
VFD_fixed_speed : BOOL;
Spare_151: BOOL;
T_Transformer_winding_temp : BOOL;
A_Transformer_winding_temp : BOOL;
T_trafo_opening_main_breaker : BOOL;
T_VFD : BOOL;
VFD_ready : BOOL;
T_VFD_emergency_stop : BOOL;
T_Low_5VDC_supply : BOOL;
T_High_5VDC_supply : BOOL;
T_Spare_9 : BOOL;
T_Spare_10 : BOOL;
T_Spare_11 : BOOL;
T_Spare_12 : BOOL;
T_Spare_13 : BOOL;
T_Low_liquid_level : BOOL;
T_SW_pump_off_to_long : BOOL;
T_Softstarter_failure : BOOL;
T_Motorstarter_failure : BOOL ;
T_CW_valveopen_failure : BOOL ;
T_SW_valveopen_failure : BOOL ;
T_High_disch_superheat :BOOL ;
T_Low_disch_superheat :BOOL ;
T_High_CW_outlet_temp : BOOL;
T_Low_CW_outlet_temp : BOOL;
T_Low_CW_inlet_temp : BOOL;
T_High_CW_inlet_temp : BOOL;
T_High_SW_outlet_temp : BOOL;
T_Low_SW_outlet_temp : BOOL;
T_Low_SW_inlet_temp : BOOL;
T_High_SW_inlet_temp : BOOL;
T_High_motor_wind_temp_R : BOOL;
T_High_motor_wind_temp_S : BOOL;
T_High_motor_wind_temp_T : BOOL;
T_High_press_ratio : BOOL;
T_Low_press_ratio : BOOL;
T_Low_CW_dP : BOOL;
T_High_CW_dP : BOOL;
T_Low_SW_dP : BOOL;
T_High_SW_dP : BOOL;
T_Long_time_PRV : BOOL;
T_Comp_thrust_neg_move : BOOL;
T_Comp_thrust_pos_move : BOOL;
T_VGD_fault : BOOL;
T_Low_oilpress_prelube : BOOL;
T_Low_temp_oil_inlet_comp : BOOL;
T_Low_oilpress_standby : BOOL;
T_Transformer : BOOL;
A_Transformer : BOOL;


T_Sensor_low_signal_AI_64 : BOOL;
T_Sensor_high_signal_AI_64 : BOOL;
T_Sensor_low_signal_AI_66 : BOOL;
T_Sensor_high_signal_AI_66 : BOOL;
T_Sensor_low_signal_AI_112 : BOOL;
T_Sensor_high_signal_AI_112 : BOOL;
T_Sensor_low_signal_AI_114 : BOOL;
T_Sensor_high_signal_AI_114 : BOOL;
T_Sensor_low_signal_AI_116 : BOOL;
T_Sensor_high_signal_AI_116 : BOOL;
T_Sensor_low_signal_AI_118 : BOOL;
T_Sensor_high_signal_AI_118 : BOOL;
T_Sensor_high_signal_AI_128 : BOOL;
T_Sensor_low_signal_AI_128 : BOOL ;
T_Sensor_high_signal_AI_130 : BOOL;
T_Sensor_low_signal_AI_130 : BOOL ;
T_Sensor_high_signal_AI_132 : BOOL;
T_Sensor_low_signal_AI_132 : BOOL ;
T_Sensor_high_signal_AI_134 : BOOL;
T_Sensor_low_signal_AI_134 : BOOL ;
T_Sensor_high_signal_AI_136 : BOOL;
T_Sensor_low_signal_AI_136 : BOOL ;
T_Sensor_high_signal_AI_138 : BOOL;
T_Sensor_low_signal_AI_138 : BOOL ;
T_Sensor_high_signal_AI_140 : BOOL;
T_Sensor_low_signal_AI_140 : BOOL ;
T_Sensor_high_signal_AI_142 : BOOL;
T_Sensor_low_signal_AI_142 : BOOL ;
T_Sensor_high_signal_AI_144 : BOOL;
T_Sensor_low_signal_AI_144 : BOOL ;
T_Sensor_high_signal_AI_146 : BOOL;
T_Sensor_low_signal_AI_146 : BOOL ;
T_Sensor_high_signal_AI_148 : BOOL;
T_Sensor_low_signal_AI_148 : BOOL ;
T_Sensor_high_signal_AI_150 : BOOL;
T_Sensor_low_signal_AI_150 : BOOL ;
T_Sensor_high_signal_AI_152 : BOOL;
T_Sensor_low_signal_AI_152 : BOOL ;
T_Sensor_high_signal_AI_154 : BOOL;
T_Sensor_low_signal_AI_154 : BOOL ;
T_Sensor_high_signal_AI_156 : BOOL;
T_Sensor_low_signal_AI_156 : BOOL ;
T_Sensor_high_signal_AI_158 : BOOL;
T_Sensor_low_signal_AI_158 : BOOL ;
T_Sensor_high_signal_AI_160 : BOOL;
T_Sensor_low_signal_AI_160 : BOOL ;
T_Sensor_high_signal_AI_162 : BOOL;
T_Sensor_low_signal_AI_162 : BOOL ;
T_Sensor_high_signal_AI_164 : BOOL;
T_Sensor_low_signal_AI_164 : BOOL ;
T_Sensor_high_signal_AI_166 : BOOL;
T_Sensor_low_signal_AI_166 : BOOL ;
T_Sensor_high_signal_AI_168 : BOOL;
T_Sensor_low_signal_AI_168 : BOOL ;
T_Sensor_high_signal_AI_170 : BOOL;
T_Sensor_low_signal_AI_170 : BOOL ;
T_Sensor_high_signal_AI_172 : BOOL;
T_Sensor_low_signal_AI_172 : BOOL ;
T_Sensor_high_signal_AI_174 : BOOL;
T_Sensor_low_signal_AI_174 : BOOL ;
T_Sensor_high_signal_AI_176 : BOOL;
T_Sensor_low_signal_AI_176 : BOOL ;
T_Sensor_low_signal_AI_178 : BOOL ;
T_Sensor_high_signal_AI_178 : BOOL;
T_Sensor_low_signal_AI_180 : BOOL ;
T_Sensor_high_signal_AI_180 : BOOL;
T_Sensor_low_signal_AI_182 : BOOL ;
T_Sensor_high_signal_AI_182 : BOOL;
T_Sensor_low_signal_AI_184 : BOOL ;
T_Sensor_high_signal_AI_184 : BOOL;
T_Sensor_low_signal_AI_186 : BOOL ;
T_Sensor_high_signal_AI_186 : BOOL;
T_Sensor_low_signal_AI_188 : BOOL ;
T_Sensor_high_signal_AI_188 : BOOL;
T_Sensor_low_signal_AI_190 : BOOL ;
T_Sensor_high_signal_AI_190 : BOOL;
T_Sensor_low_signal_AI_192 : BOOL ;
T_Sensor_high_signal_AI_192 : BOOL;
T_Sensor_low_signal_AI_194 : BOOL ;
T_Sensor_high_signal_AI_194 : BOOL;
T_Sensor_low_signal_AI_196 : BOOL ;
T_Sensor_high_signal_AI_196 : BOOL;
T_Sensor_low_signal_AI_198 : BOOL ;
T_Sensor_high_signal_AI_198 : BOOL;
T_Sensor_high_signal_AI_200 : BOOL;
T_Sensor_low_signal_AI_200 : BOOL ;
T_Sensor_low_signal_AI_202 : BOOL ;
T_Sensor_high_signal_AI_202 : BOOL;
T_Sensor_low_signal_AI_204 : BOOL ;
T_Sensor_high_signal_AI_204 : BOOL;
T_Sensor_low_signal_AI_206 : BOOL ;
T_Sensor_high_signal_AI_206 : BOOL ;
CW_Pump_Remote_Start_Available : BOOL;
T_CW_Pump : BOOL;
A_high_disch_press : BOOL ;
A_low_disch_press : BOOL ;
A_Low_suction_pressure : BOOL;
A_High_suction_pressure : BOOL;
A_High_discharge_temp : BOOL;
A_High_oil_temp_receiver : BOOL;
A_Low_oil_temp_receiver : BOOL;
A_Low_temp_oil_inlet_comp : BOOL;
A_High_oil_diff_pressure : BOOL;
A_Low_discharge_superheat : BOOL;
A_High_discharge_superheat : BOOL;
A_Low_CW_outlet_temp : BOOL;
A_High_CW_outlet_temp : BOOL;
A_Low_CW_inlet_temp : BOOL;
A_High_CW_inlet_temp : BOOL;
A_High_SW_outlet_temp : BOOL;
A_Low_condenser_flow : BOOL;
A_High_press_ratio : BOOL;
A_Low_press_ratio : BOOL;
A_Motor_speed_low : BOOL;
A_Low_SW_outlet_temp : BOOL;
A_Low_SW_inlet_temp : BOOL;
A_High_SW_inlet_temp : BOOL;
A_High_suction_superheat : BOOL;
A_Low_suction_superheat : BOOL;
A_High_temp_oil_separator : BOOL;
A_Low_temp_oil_separator : BOOL;
A_High_motor_wind_temp_R : BOOL;
A_High_motor_wind_temp_S : BOOL;
A_High_motor_wind_temp_T : BOOL;
A_High_CW_dP : BOOL;
A_Low_CW_dP : BOOL;
A_High_SW_dP : BOOL;
A_Low_SW_dP : BOOL;
A_VGD_Fault : BOOL;
Start_inhib_time_between_Start : BOOL;
Start_inhib_time_between_Stop_Start : BOOL;
Start_inhib_PRV_not_min : BOOL;
Start_inhib_Motor_overload : BOOL;
Remote_bilge_pump_control : BOOL;
CW_pump_running : BOOL;
A_Low_liquid_level : BOOL;
A_Suction_press_limit : BOOL;
A_Discharge_press_limit : BOOL;
A_Discharge_superheat_limit : BOOL;
A_Motor_current_limit : BOOL;


DI_0_0_Emergency_stop : BOOL;
DI_0_1 : BOOL;
DI_0_2_Fault_reset : BOOL;
DI_0_3 : BOOL;
DI_0_4 : BOOL;
DI_0_5 : BOOL;
DI_0_6_Overload_protection : BOOL;
DI_0_7 : BOOL;
DI_1_0_Overload_oilpump : BOOL;
DI_1_1 : BOOL;
DI_1_2 : BOOL;
DI_1_3 : BOOL;
DI_1_4_Power_available : BOOL;
DI_1_5_Starter_failure : BOOL;
DI_8_0_Controlpanel_temp : BOOL;
DI_8_1 : BOOL;
DI_8_2_VGD_limit_switch : BOOL;
DI_8_3_water_leak_motor  : BOOL;
DI_8_4_Catodic_protection : BOOL;
DI_8_5_Trust_bearing_probe : BOOL;
DI_8_6_ESD_operation : BOOL;
DI_8_7 : BOOL;
DI_9_0_MV_breaker_available : BOOL;
DI_9_1 : BOOL;
DI_9_2_Safe_return_to_port : BOOL;
DI_9_3 : BOOL;
DI_9_4_VFD_emergency_stop : BOOL;
DI_9_5 : BOOL;
DI_9_6 : BOOL;
DI_9_7 : BOOL;
DO_0_0_Start_signal_comp : BOOL;
DO_0_1_Start_signal_oil_pump : BOOL;
DO_0_2_Start_signal_SW_pump : BOOL;
DO_0_3_Start_signal_CW_pump : BOOL;
DO_0_4_Solenoid_valve_oil : BOOL;
DO_0_5_Solenoid_valve_liquid : BOOL;
DO_0_6_Oil_heater : BOOL;
DO_0_7_Comp_heater : BOOL;
DO_1_0 : BOOL;
DO_1_1 : BOOL;
DO_8_0_Liquid_valve_open : BOOL;
DO_8_1_Liquid_valve_close : BOOL;
DO_8_2_VGD_open : BOOL;
DO_8_3_VGD_close : BOOL;
DO_8_4_PRV_open : BOOL;
DO_8_5_PRV_close : BOOL;
DO_8_6_HGV_open : BOOL;
DO_8_7_HGV_close : BOOL;
DO_9_0_Main_breaker_ready : BOOL;
DO_9_1_Close_order_swv_overboard : BOOL;
DO_9_2_Open_order_swv_bypass : BOOL;
DO_9_3_Close_order_swv_bypass : BOOL;
DO_9_4 : BOOL;
DO_9_5 : BOOL;
DO_9_6 : BOOL;
DO_9_7 : BOOL;
DO_12_0_Power_request : BOOL;
DO_12_1_Compressor_ready : BOOL;
DO_12_2 : BOOL;
DO_12_3 : BOOL;
DO_12_4_Control_panel_alarm : BOOL;
DO_12_5_Auto_reset : BOOL;
DO_12_6_Unit_running : BOOL;
DO_12_7_Emergency_MV_Breaker : BOOL;
Start_inhib_time_Oil_receiver_temp : BOOL;



//Graphic variables
Unit_switch_status : INT;
i : INT;
show_trendvalue : ARRAY[0..50] OF BOOL;
select_trendvalue : INT :=0 ;

END_VAR

